LIN {X 0,Y 468.13,Z 261.484,A -85,B 0,C 180,E1 -7681.158,E2 -7681.158} C_VEL
LIN {X 0,Y 468.441,Z 256.136,A -85,B 0,C 180,E1 -7683.717,E2 -7683.717} C_VEL
LIN {X 0,Y 468.542,Z 251.799,A -85,B 0,C 180,E1 -7685.905,E2 -7685.905} C_VEL
LIN {X 0,Y 468.023,Z 247.93,A -85,B 0,C 180,E1 -7688,E2 -7688} C_VEL
LIN {X 0,Y 467.596,Z 245.244,A -85,B 0,C 180,E1 -7689.56,E2 -7689.56} C_VEL
LIN {X 0,Y 467.586,Z 245.243,A -85,B 0,C 180,E1 -7692.566,E2 -7692.566} C_VEL
LIN {X 0,Y 467.569,Z 245.245,A -85,B 0,C 180,E1 -7695.052,E2 -7695.052} C_VEL
LIN {X 0,Y 467.587,Z 245.245,A -85,B 0,C 180,E1 -7697.439,E2 -7697.439} C_VEL
LIN {X 0,Y 467.613,Z 245.241,A -85,B 0,C 180,E1 -7700.857,E2 -7700.857} C_VEL
LIN {X 0,Y 467.561,Z 245.245,A -85,B 0,C 180,E1 -7704.259,E2 -7704.259} C_VEL
LIN {X 0,Y 467.579,Z 245.243,A -85,B 0,C 180,E1 -7707.32,E2 -7707.32} C_VEL
LIN {X 0,Y 467.574,Z 245.244,A -85,B 0,C 180,E1 -7710.664,E2 -7710.664} C_VEL
LIN {X 0,Y 467.612,Z 245.239,A -85,B 0,C 180,E1 -7713.199,E2 -7713.199} C_VEL
LIN {X 0,Y 467.588,Z 245.242,A -85,B 0,C 180,E1 -7716.467,E2 -7716.467} C_VEL
LIN {X 0,Y 467.617,Z 245.239,A -85,B 0,C 180,E1 -7719.776,E2 -7719.776} C_VEL
LIN {X 0,Y 467.603,Z 245.24,A -85,B 0,C 180,E1 -7722.506,E2 -7722.506} C_VEL
LIN {X 0,Y 467.6,Z 245.242,A -85,B 0,C 180,E1 -7725.195,E2 -7725.195} C_VEL
LIN {X 0,Y 467.65,Z 245.234,A -85,B 0,C 180,E1 -7727.853,E2 -7727.853} C_VEL
LIN {X 0,Y 467.676,Z 245.232,A -85,B 0,C 180,E1 -7731.356,E2 -7731.356} C_VEL
LIN {X 0,Y 467.737,Z 245.224,A -85,B 0,C 180,E1 -7733.962,E2 -7733.962} C_VEL
LIN {X 0,Y 467.852,Z 245.21,A -85,B 0,C 180,E1 -7737.416,E2 -7737.416} C_VEL
LIN {X 0,Y 467.874,Z 245.207,A -85,B 0,C 180,E1 -7739.999,E2 -7739.999} C_VEL
LIN {X 0,Y 467.853,Z 245.211,A -85,B 0,C 180,E1 -7742.582,E2 -7742.582} C_VEL
LIN {X 0,Y 467.735,Z 245.225,A -85,B 0,C 180,E1 -7746.036,E2 -7746.036} C_VEL
LIN {X 0,Y 467.667,Z 245.234,A -85,B 0,C 180,E1 -7748.642,E2 -7748.642} C_VEL
LIN {X 0,Y 467.605,Z 245.241,A -85,B 0,C 180,E1 -7749.515,E2 -7749.515} C_VEL
LIN {X 0,Y 467.573,Z 245.747,A -85,B 0,C 180,E1 -7750.39,E2 -7750.39} C_VEL
LIN {X 0,Y 467.64,Z 248.338,A -85,B 0,C 180,E1 -7752.355,E2 -7752.355} C_VEL
LIN {X 0,Y 467.428,Z 253.066,A -85,B 0,C 180,E1 -7755.793,E2 -7755.793} C_VEL
LIN {X 0,Y 467.31,Z 257.112,A -85,B 0,C 180,E1 -7758.657,E2 -7758.657} C_VEL
LIN {X 0,Y 467.115,Z 262.092,A -85,B 0,C 180,E1 -7762.093,E2 -7762.093} C_VEL
LIN {X 0,Y 467.018,Z 267.081,A -85,B 0,C 180,E1 -7765.458,E2 -7765.458} C_VEL
LIN {X 0,Y 466.893,Z 270.645,A -85,B 0,C 180,E1 -7767.815,E2 -7767.815} C_VEL
LIN {X 0,Y 466.818,Z 275.003,A -85,B 0,C 180,E1 -7770.662,E2 -7770.662} C_VEL
LIN {X 0,Y 469.826,Z 289.237,A -85,B 0,C 180,E1 -7771.206,E2 -7771.206} C_VEL
LIN {X 0,Y 470.243,Z 292.705,A -85,B 0,C 180,E1 -7771.356,E2 -7771.356} C_VEL
LIN {X 0,Y 469.793,Z 305.072,A -85,B 0,C 180,E1 -7771.95,E2 -7771.95} C_VEL
LIN {X 0,Y 469.318,Z 316.987,A -85,B 0,C 180,E1 -7772.707,E2 -7772.707} C_VEL
LIN {X 0,Y 468.82,Z 327.819,A -85,B 0,C 180,E1 -7773.59,E2 -7773.59} C_VEL
LIN {X 0,Y 468.31,Z 338.331,A -85,B 0,C 180,E1 -7774.658,E2 -7774.658} C_VEL
LIN {X 0,Y 467.835,Z 347.892,A -85,B 0,C 180,E1 -7775.863,E2 -7775.863} C_VEL
LIN {X 0,Y 467.428,Z 356.162,A -85,B 0,C 180,E1 -7777.169,E2 -7777.169} C_VEL
LIN {X 0,Y 467.115,Z 363.055,A -85,B 0,C 180,E1 -7778.524,E2 -7778.524} C_VEL
LIN {X 0,Y 466.89,Z 368.416,A -85,B 0,C 180,E1 -7779.854,E2 -7779.854} C_VEL
LIN {X 0,Y 466.773,Z 372.503,A -85,B 0,C 180,E1 -7781.165,E2 -7781.165} C_VEL
LIN {X 0,Y 466.611,Z 375.893,A -85,B 0,C 180,E1 -7782.669,E2 -7782.669} C_VEL
LIN {X 0,Y 466.534,Z 377.66,A -85,B 0,C 180,E1 -7783.863,E2 -7783.863} C_VEL
LIN {X 0,Y 466.558,Z 378.644,A -85,B 0,C 180,E1 -7785.069,E2 -7785.069} C_VEL
LIN {X 0,Y 466.498,Z 378.866,A -85,B 0,C 180,E1 -7786.312,E2 -7786.312} C_VEL
LIN {X 0,Y 466.518,Z 378.258,A -85,B 0,C 180,E1 -7787.574,E2 -7787.574} C_VEL
LIN {X 0,Y 466.585,Z 376.759,A -85,B 0,C 180,E1 -7788.86,E2 -7788.86} C_VEL
LIN {X 0,Y 466.664,Z 374.263,A -85,B 0,C 180,E1 -7790.178,E2 -7790.178} C_VEL
LIN {X 0,Y 466.84,Z 370.669,A -85,B 0,C 180,E1 -7791.518,E2 -7791.518} C_VEL
LIN {X 0,Y 466.998,Z 365.358,A -85,B 0,C 180,E1 -7792.99,E2 -7792.99} C_VEL
LIN {X 0,Y 467.311,Z 358.15,A -85,B 0,C 180,E1 -7794.524,E2 -7794.524} C_VEL
LIN {X 0,Y 467.631,Z 350.889,A -85,B 0,C 180,E1 -7795.748,E2 -7795.748} C_VEL
LIN {X 0,Y 468.119,Z 341.5,A -85,B 0,C 180,E1 -7797.019,E2 -7797.019} C_VEL
LIN {X 0,Y 468.575,Z 331.818,A -85,B 0,C 180,E1 -7798.083,E2 -7798.083} C_VEL
LIN {X 0,Y 469.009,Z 321.069,A -85,B 0,C 180,E1 -7799.036,E2 -7799.036} C_VEL
LIN {X 0,Y 469.461,Z 309.708,A -85,B 0,C 180,E1 -7799.833,E2 -7799.833} C_VEL
LIN {X 0,Y 469.96,Z 297.671,A -85,B 0,C 180,E1 -7800.485,E2 -7800.485} C_VEL
LIN {X 0,Y 469.928,Z 290.386,A -85,B 0,C 180,E1 -7800.802,E2 -7800.802} C_VEL
LIN {X 0,Y 468.566,Z 283.472,A -85,B 0,C 180,E1 -7801.088,E2 -7801.088} C_VEL
LIN {X 0,Y 467.583,Z 280.229,A -85,B 0,C 180,E1 -7801.292,E2 -7801.292} C_VEL
LIN {X 0,Y 466.265,Z 277.641,A -85,B 0,C 180,E1 -7801.595,E2 -7801.595} C_VEL
LIN {X 0,Y 464.069,Z 274.82,A -85,B 0,C 180,E1 -7802.168,E2 -7802.168} C_VEL
LIN {X 0,Y 461.965,Z 272.984,A -85,B 0,C 180,E1 -7802.848,E2 -7802.848} C_VEL
LIN {X 0,Y 460.022,Z 271.336,A -85,B 0,C 180,E1 -7803.841,E2 -7803.841} C_VEL
LIN {X 0,Y 459.75,Z 270.573,A -85,B 0,C 180,E1 -7804.353,E2 -7804.353} C_VEL
LIN {X 0,Y 459.891,Z 265.717,A -85,B 0,C 180,E1 -7807.54,E2 -7807.54} C_VEL
LIN {X 0,Y 460.007,Z 261.493,A -85,B 0,C 180,E1 -7810.36,E2 -7810.36} C_VEL
LIN {X 0,Y 460.108,Z 257.409,A -85,B 0,C 180,E1 -7813.129,E2 -7813.129} C_VEL
LIN {X 0,Y 460.211,Z 253.466,A -85,B 0,C 180,E1 -7815.858,E2 -7815.858} C_VEL
LIN {X 0,Y 460.408,Z 249.613,A -85,B 0,C 180,E1 -7818.555,E2 -7818.555} C_VEL
LIN {X 0,Y 460.473,Z 246.127,A -85,B 0,C 180,E1 -7821.221,E2 -7821.221} C_VEL
LIN {X 0,Y 460.692,Z 246.1,A -85,B 0,C 180,E1 -7823.87,E2 -7823.87} C_VEL
LIN {X 0,Y 460.814,Z 246.084,A -85,B 0,C 180,E1 -7827.378,E2 -7827.378} C_VEL
LIN {X 0,Y 460.842,Z 246.082,A -85,B 0,C 180,E1 -7830,E2 -7830} C_VEL
LIN {X 0,Y 460.816,Z 246.086,A -85,B 0,C 180,E1 -7832.622,E2 -7832.622} C_VEL
LIN {X 0,Y 460.7,Z 246.1,A -85,B 0,C 180,E1 -7836.13,E2 -7836.13} C_VEL
LIN {X 0,Y 460.619,Z 246.11,A -85,B 0,C 180,E1 -7838.776,E2 -7838.776} C_VEL
LIN {X 0,Y 460.623,Z 246.11,A -85,B 0,C 180,E1 -7842.457,E2 -7842.457} C_VEL
LIN {X 0,Y 460.611,Z 246.111,A -85,B 0,C 180,E1 -7846.007,E2 -7846.007} C_VEL
LIN {X 0,Y 460.559,Z 246.117,A -85,B 0,C 180,E1 -7849.616,E2 -7849.616} C_VEL
LIN {X 0,Y 460.519,Z 246.122,A -85,B 0,C 180,E1 -7852.428,E2 -7852.428} C_VEL
LIN {X 0,Y 460.558,Z 246.118,A -85,B 0,C 180,E1 -7855.803,E2 -7855.803} C_VEL
LIN {X 0,Y 460.547,Z 246.12,A -85,B 0,C 180,E1 -7858.233,E2 -7858.233} C_VEL
LIN {X 0,Y 460.514,Z 246.123,A -85,B 0,C 180,E1 -7861.284,E2 -7861.284} C_VEL
LIN {X 0,Y 460.523,Z 246.121,A -85,B 0,C 180,E1 -7864.506,E2 -7864.506} C_VEL
LIN {X 0,Y 460.52,Z 246.123,A -85,B 0,C 180,E1 -7867.621,E2 -7867.621} C_VEL
LIN {X 0,Y 460.549,Z 246.118,A -85,B 0,C 180,E1 -7870.273,E2 -7870.273} C_VEL
LIN {X 0,Y 460.514,Z 246.123,A -85,B 0,C 180,E1 -7873.373,E2 -7873.373} C_VEL
LIN {X 0,Y 460.514,Z 246.123,A -85,B 0,C 180,E1 -7876.628,E2 -7876.628} C_VEL
LIN {X 0,Y 460.549,Z 246.12,A -85,B 0,C 180,E1 -7879.728,E2 -7879.728} C_VEL
LIN {X 0,Y 460.518,Z 246.122,A -85,B 0,C 180,E1 -7882.52,E2 -7882.52} C_VEL
LIN {X 0,Y 460.538,Z 246.12,A -85,B 0,C 180,E1 -7885.625,E2 -7885.625} C_VEL
LIN {X 0,Y 460.526,Z 246.122,A -85,B 0,C 180,E1 -7888.745,E2 -7888.745} C_VEL
LIN {X 0,Y 460.548,Z 246.118,A -85,B 0,C 180,E1 -7891.768,E2 -7891.768} C_VEL
LIN {X 0,Y 460.55,Z 246.12,A -85,B 0,C 180,E1 -7894.706,E2 -7894.706} C_VEL
LIN {X 0,Y 460.503,Z 246.124,A -85,B 0,C 180,E1 -7897.572,E2 -7897.572} C_VEL
LIN {X 0,Y 460.56,Z 246.117,A -85,B 0,C 180,E1 -7900.385,E2 -7900.385} C_VEL
LIN {X 0,Y 460.557,Z 246.117,A -85,B 0,C 180,E1 -7903.147,E2 -7903.147} C_VEL
LIN {X 0,Y 460.545,Z 246.117,A -85,B 0,C 180,E1 -7905.869,E2 -7905.869} C_VEL
LIN {X 0,Y 460.605,Z 246.113,A -85,B 0,C 180,E1 -7908.56,E2 -7908.56} C_VEL
LIN {X 0,Y 460.688,Z 246.101,A -85,B 0,C 180,E1 -7912.11,E2 -7912.11} C_VEL
LIN {X 0,Y 460.691,Z 246.102,A -85,B 0,C 180,E1 -7914.749,E2 -7914.749} C_VEL
LIN {X 0,Y 460.818,Z 246.084,A -85,B 0,C 180,E1 -7917.379,E2 -7917.379} C_VEL
LIN {X 0,Y 460.845,Z 246.082,A -85,B 0,C 180,E1 -7920.001,E2 -7920.001} C_VEL
LIN {X 0,Y 460.819,Z 246.085,A -85,B 0,C 180,E1 -7922.623,E2 -7922.623} C_VEL
LIN {X 0,Y 460.704,Z 246.1,A -85,B 0,C 180,E1 -7926.131,E2 -7926.131} C_VEL
LIN {X 0,Y 460.623,Z 246.109,A -85,B 0,C 180,E1 -7928.777,E2 -7928.777} C_VEL
LIN {X 0,Y 460.63,Z 246.109,A -85,B 0,C 180,E1 -7932.458,E2 -7932.458} C_VEL
LIN {X 0,Y 460.596,Z 246.113,A -85,B 0,C 180,E1 -7935.999,E2 -7935.999} C_VEL
LIN {X 0,Y 460.567,Z 246.116,A -85,B 0,C 180,E1 -7938.903,E2 -7938.903} C_VEL
LIN {X 0,Y 460.512,Z 246.124,A -85,B 0,C 180,E1 -7941.487,E2 -7941.487} C_VEL
LIN {X 0,Y 460.539,Z 246.119,A -85,B 0,C 180,E1 -7944.333,E2 -7944.333} C_VEL
LIN {X 0,Y 460.57,Z 246.117,A -85,B 0,C 180,E1 -7947.245,E2 -7947.245} C_VEL
LIN {X 0,Y 460.508,Z 246.122,A -85,B 0,C 180,E1 -7950.241,E2 -7950.241} C_VEL
LIN {X 0,Y 460.525,Z 246.123,A -85,B 0,C 180,E1 -7953.326,E2 -7953.326} C_VEL
LIN {X 0,Y 460.477,Z 246.126,A -85,B 0,C 180,E1 -7956.53,E2 -7956.53} C_VEL
LIN {X 0,Y 460.544,Z 246.119,A -85,B 0,C 180,E1 -7958.899,E2 -7958.899} C_VEL
LIN {X 0,Y 460.522,Z 246.119,A -85,B 0,C 180,E1 -7962.182,E2 -7962.182} C_VEL
LIN {X 0,Y 460.514,Z 246.123,A -85,B 0,C 180,E1 -7965.412,E2 -7965.412} C_VEL
LIN {X 0,Y 460.533,Z 246.12,A -85,B 0,C 180,E1 -7968.398,E2 -7968.398} C_VEL
LIN {X 0,Y 460.573,Z 246.124,A -85,B 0,C 180,E1 -7970.78,E2 -7970.78} C_VEL
LIN {X 0,Y 461.389,Z 251.451,A -85,B 0,C 180,E1 -7973.555,E2 -7973.555} C_VEL
LIN {X 0,Y 461.454,Z 255.827,A -85,B 0,C 180,E1 -7975.701,E2 -7975.701} C_VEL
LIN {X 0,Y 461.128,Z 262.38,A -85,B 0,C 180,E1 -7978.79,E2 -7978.79} C_VEL
LIN {X 0,Y 460.758,Z 268.954,A -85,B 0,C 180,E1 -7981.781,E2 -7981.781} C_VEL
LIN {X 0,Y 460.48,Z 276.639,A -85,B 0,C 180,E1 -7985.184,E2 -7985.184} C_VEL
LIN {X 0,Y 460.243,Z 284.73,A -85,B 0,C 180,E1 -7988.668,E2 -7988.668} C_VEL
LIN {X 0,Y 460.03,Z 292.037,A -85,B 0,C 180,E1 -7991.749,E2 -7991.749} C_VEL
LIN {X 0,Y 459.886,Z 298.398,A -85,B 0,C 180,E1 -7994.387,E2 -7994.387} C_VEL
LIN {X 0,Y 462.114,Z 312.279,A -85,B 0,C 180,E1 -7994.853,E2 -7994.853} C_VEL
LIN {X 0,Y 463.006,Z 320.585,A -85,B 0,C 180,E1 -7995.215,E2 -7995.215} C_VEL
LIN {X 0,Y 462.542,Z 332.447,A -85,B 0,C 180,E1 -7995.818,E2 -7995.818} C_VEL
LIN {X 0,Y 462.017,Z 343.944,A -85,B 0,C 180,E1 -7996.587,E2 -7996.587} C_VEL
LIN {X 0,Y 461.494,Z 355.106,A -85,B 0,C 180,E1 -7997.533,E2 -7997.533} C_VEL
LIN {X 0,Y 461.029,Z 364.99,A -85,B 0,C 180,E1 -7998.57,E2 -7998.57} C_VEL
LIN {X 0,Y 460.508,Z 373.569,A -85,B 0,C 180,E1 -7999.67,E2 -7999.67} C_VEL
LIN {X 0,Y 460.148,Z 381.911,A -85,B 0,C 180,E1 -8000.993,E2 -8000.993} C_VEL
LIN {X 0,Y 459.889,Z 388.636,A -85,B 0,C 180,E1 -8002.316,E2 -8002.316} C_VEL
LIN {X 0,Y 459.666,Z 394.798,A -85,B 0,C 180,E1 -8003.856,E2 -8003.856} C_VEL
LIN {X 0,Y 459.618,Z 398.796,A -85,B 0,C 180,E1 -8005.176,E2 -8005.176} C_VEL
LIN {X 0,Y 459.584,Z 401.745,A -85,B 0,C 180,E1 -8006.493,E2 -8006.493} C_VEL
LIN {X 0,Y 459.585,Z 403.152,A -85,B 0,C 180,E1 -8007.37,E2 -8007.37} C_VEL
LIN {X 0,Y 459.522,Z 404.758,A -85,B 0,C 180,E1 -8009.124,E2 -8009.124} C_VEL
LIN {X 0,Y 459.53,Z 404.974,A -85,B 0,C 180,E1 -8010,E2 -8010} C_VEL
LIN {X 0,Y 459.522,Z 404.753,A -85,B 0,C 180,E1 -8010.876,E2 -8010.876} C_VEL
LIN {X 0,Y 459.585,Z 403.129,A -85,B 0,C 180,E1 -8012.629,E2 -8012.629} C_VEL
LIN {X 0,Y 459.584,Z 401.718,A -85,B 0,C 180,E1 -8013.507,E2 -8013.507} C_VEL
LIN {X 0,Y 459.618,Z 398.753,A -85,B 0,C 180,E1 -8014.824,E2 -8014.824} C_VEL
LIN {X 0,Y 459.716,Z 393.705,A -85,B 0,C 180,E1 -8016.431,E2 -8016.431} C_VEL
LIN {X 0,Y 459.908,Z 387.566,A -85,B 0,C 180,E1 -8017.905,E2 -8017.905} C_VEL
LIN {X 0,Y 460.224,Z 380.617,A -85,B 0,C 180,E1 -8019.227,E2 -8019.227} C_VEL
LIN {X 0,Y 460.593,Z 371.922,A -85,B 0,C 180,E1 -8020.55,E2 -8020.55} C_VEL
LIN {X 0,Y 461.119,Z 363.024,A -85,B 0,C 180,E1 -8021.65,E2 -8021.65} C_VEL
LIN {X 0,Y 461.567,Z 352.267,A -85,B 0,C 180,E1 -8022.738,E2 -8022.738} C_VEL
LIN {X 0,Y 462.138,Z 341.06,A -85,B 0,C 180,E1 -8023.634,E2 -8023.634} C_VEL
LIN {X 0,Y 462.756,Z 328.773,A -85,B 0,C 180,E1 -8024.4,E2 -8024.4} C_VEL
LIN {X 0,Y 462.968,Z 318.49,A -85,B 0,C 180,E1 -8024.899,E2 -8024.899} C_VEL
LIN {X 0,Y 461.165,Z 305.618,A -85,B 0,C 180,E1 -8025.425,E2 -8025.425} C_VEL
LIN {X 0,Y 459.851,Z 297.977,A -85,B 0,C 180,E1 -8025.666,E2 -8025.666} C_VEL
LIN {X 0,Y 460.014,Z 290.618,A -85,B 0,C 180,E1 -8028.713,E2 -8028.713} C_VEL
LIN {X 0,Y 460.265,Z 282.926,A -85,B 0,C 180,E1 -8031.968,E2 -8031.968} C_VEL
LIN {X 0,Y 460.504,Z 275.275,A -85,B 0,C 180,E1 -8035.297,E2 -8035.297} C_VEL
LIN {X 0,Y 460.784,Z 267.719,A -85,B 0,C 180,E1 -8038.714,E2 -8038.714} C_VEL
LIN {X 0,Y 461.147,Z 262.006,A -85,B 0,C 180,E1 -8041.41,E2 -8041.41} C_VEL
LIN {X 0,Y 461.529,Z 255.372,A -85,B 0,C 180,E1 -8044.684,E2 -8044.684} C_VEL
LIN {X 0,Y 461.354,Z 251.017,A -85,B 0,C 180,E1 -8046.992,E2 -8046.992} C_VEL
LIN {X 0,Y 460.562,Z 246.12,A -85,B 0,C 180,E1 -8049.858,E2 -8049.858} C_VEL
LIN {X 0,Y 460.516,Z 246.123,A -85,B 0,C 180,E1 -8052.9,E2 -8052.9} C_VEL
LIN {X 0,Y 460.51,Z 246.125,A -85,B 0,C 180,E1 -8055.829,E2 -8055.829} C_VEL
LIN {X 0,Y 460.537,Z 246.123,A -85,B 0,C 180,E1 -8058.989,E2 -8058.989} C_VEL
LIN {X 0,Y 460.542,Z 246.121,A -85,B 0,C 180,E1 -8061.268,E2 -8061.268} C_VEL
LIN {X 0,Y 460.511,Z 246.125,A -85,B 0,C 180,E1 -8064.554,E2 -8064.554} C_VEL
LIN {X 0,Y 460.529,Z 246.122,A -85,B 0,C 180,E1 -8067.715,E2 -8067.715} C_VEL
LIN {X 0,Y 460.543,Z 246.121,A -85,B 0,C 180,E1 -8070.768,E2 -8070.768} C_VEL
LIN {X 0,Y 460.558,Z 246.118,A -85,B 0,C 180,E1 -8073.734,E2 -8073.734} C_VEL
LIN {X 0,Y 460.541,Z 246.12,A -85,B 0,C 180,E1 -8076.623,E2 -8076.623} C_VEL
LIN {X 0,Y 460.545,Z 246.12,A -85,B 0,C 180,E1 -8079.452,E2 -8079.452} C_VEL
LIN {X 0,Y 460.554,Z 246.119,A -85,B 0,C 180,E1 -8082.229,E2 -8082.229} C_VEL
LIN {X 0,Y 460.559,Z 246.118,A -85,B 0,C 180,E1 -8084.964,E2 -8084.964} C_VEL
LIN {X 0,Y 460.607,Z 246.112,A -85,B 0,C 180,E1 -8088.558,E2 -8088.558} C_VEL
LIN {X 0,Y 460.688,Z 246.102,A -85,B 0,C 180,E1 -8092.107,E2 -8092.107} C_VEL
LIN {X 0,Y 460.691,Z 246.1,A -85,B 0,C 180,E1 -8094.747,E2 -8094.747} C_VEL
LIN {X 0,Y 460.817,Z 246.086,A -85,B 0,C 180,E1 -8097.377,E2 -8097.377} C_VEL
LIN {X 0,Y 460.844,Z 246.082,A -85,B 0,C 180,E1 -8099.999,E2 -8099.999} C_VEL
LIN {X 0,Y 460.818,Z 246.088,A -85,B 0,C 180,E1 -8102.621,E2 -8102.621} C_VEL
LIN {X 0,Y 460.701,Z 246.101,A -85,B 0,C 180,E1 -8106.129,E2 -8106.129} C_VEL
LIN {X 0,Y 460.608,Z 246.114,A -85,B 0,C 180,E1 -8108.775,E2 -8108.775} C_VEL
LIN {X 0,Y 460.559,Z 246.119,A -85,B 0,C 180,E1 -8109.662,E2 -8109.662} C_VEL
LIN {X 0,Y 460.61,Z 248.118,A -85,B 0,C 180,E1 -8111.44,E2 -8111.44} C_VEL
LIN {X 0,Y 460.456,Z 251.718,A -85,B 0,C 180,E1 -8114.134,E2 -8114.134} C_VEL
LIN {X 0,Y 460.322,Z 255.431,A -85,B 0,C 180,E1 -8116.862,E2 -8116.862} C_VEL
LIN {X 0,Y 460.157,Z 259.349,A -85,B 0,C 180,E1 -8119.632,E2 -8119.632} C_VEL
LIN {X 0,Y 460.055,Z 263.387,A -85,B 0,C 180,E1 -8122.451,E2 -8122.451} C_VEL
LIN {X 0,Y 459.94,Z 268.062,A -85,B 0,C 180,E1 -8125.642,E2 -8125.642} C_VEL
LIN {X 0,Y 459.777,Z 272.019,A -85,B 0,C 180,E1 -8128.283,E2 -8128.283} C_VEL
LIN {X 0,Y 459.746,Z 275.371,A -85,B 0,C 180,E1 -8130.421,E2 -8130.421} C_VEL
LIN {X 0,Y 462.665,Z 288.74,A -85,B 0,C 180,E1 -8130.935,E2 -8130.935} C_VEL
LIN {X 0,Y 463.395,Z 293.049,A -85,B 0,C 180,E1 -8131.133,E2 -8131.133} C_VEL
LIN {X 0,Y 462.905,Z 305.934,A -85,B 0,C 180,E1 -8131.767,E2 -8131.767} C_VEL
LIN {X 0,Y 462.415,Z 317.503,A -85,B 0,C 180,E1 -8132.522,E2 -8132.522} C_VEL
LIN {X 0,Y 461.879,Z 328.845,A -85,B 0,C 180,E1 -8133.474,E2 -8133.474} C_VEL
LIN {X 0,Y 461.349,Z 338.478,A -85,B 0,C 180,E1 -8134.473,E2 -8134.473} C_VEL
LIN {X 0,Y 460.829,Z 348.261,A -85,B 0,C 180,E1 -8135.727,E2 -8135.727} C_VEL
LIN {X 0,Y 460.42,Z 356.115,A -85,B 0,C 180,E1 -8136.983,E2 -8136.983} C_VEL
LIN {X 0,Y 460.093,Z 362.404,A -85,B 0,C 180,E1 -8138.215,E2 -8138.215} C_VEL
LIN {X 0,Y 459.871,Z 368.214,A -85,B 0,C 180,E1 -8139.644,E2 -8139.644} C_VEL
LIN {X 0,Y 459.687,Z 372.748,A -85,B 0,C 180,E1 -8141.101,E2 -8141.101} C_VEL
LIN {X 0,Y 459.527,Z 376.351,A -85,B 0,C 180,E1 -8142.769,E2 -8142.769} C_VEL
LIN {X 0,Y 459.443,Z 378.086,A -85,B 0,C 180,E1 -8144.034,E2 -8144.034} C_VEL
LIN {X 0,Y 459.453,Z 378.969,A -85,B 0,C 180,E1 -8145.282,E2 -8145.282} C_VEL
LIN {X 0,Y 459.405,Z 379.03,A -85,B 0,C 180,E1 -8146.497,E2 -8146.497} C_VEL
LIN {X 0,Y 459.422,Z 378.362,A -85,B 0,C 180,E1 -8147.695,E2 -8147.695} C_VEL
LIN {X 0,Y 459.494,Z 376.99,A -85,B 0,C 180,E1 -8148.877,E2 -8148.877} C_VEL
LIN {X 0,Y 459.628,Z 373.546,A -85,B 0,C 180,E1 -8150.614,E2 -8150.614} C_VEL
LIN {X 0,Y 459.838,Z 368.499,A -85,B 0,C 180,E1 -8152.314,E2 -8152.314} C_VEL
LIN {X 0,Y 460.06,Z 362.624,A -85,B 0,C 180,E1 -8153.77,E2 -8153.77} C_VEL
LIN {X 0,Y 460.372,Z 356.11,A -85,B 0,C 180,E1 -8155.052,E2 -8155.052} C_VEL
LIN {X 0,Y 460.711,Z 349.207,A -85,B 0,C 180,E1 -8156.166,E2 -8156.166} C_VEL
LIN {X 0,Y 461.226,Z 340.032,A -85,B 0,C 180,E1 -8157.383,E2 -8157.383} C_VEL
LIN {X 0,Y 461.657,Z 329.713,A -85,B 0,C 180,E1 -8158.483,E2 -8158.483} C_VEL
LIN {X 0,Y 462.192,Z 319.286,A -85,B 0,C 180,E1 -8159.377,E2 -8159.377} C_VEL
LIN {X 0,Y 462.64,Z 307.799,A -85,B 0,C 180,E1 -8160.166,E2 -8160.166} C_VEL
LIN {X 0,Y 463.149,Z 296.398,A -85,B 0,C 180,E1 -8160.764,E2 -8160.764} C_VEL
LIN {X 0,Y 463.003,Z 291.008,A -85,B 0,C 180,E1 -8161.002,E2 -8161.002} C_VEL
LIN {X 0,Y 460.244,Z 277.687,A -85,B 0,C 180,E1 -8161.53,E2 -8161.53} C_VEL
LIN {X 0,Y 459.698,Z 274.743,A -85,B 0,C 180,E1 -8161.648,E2 -8161.648} C_VEL
LIN {X 0,Y 459.75,Z 270.573,A -85,B 0,C 180,E1 -8164.353,E2 -8164.353} C_VEL
LIN {X 0,Y 459.134,Z 269.529,A -85,B 0,C 180,E1 -8165.073,E2 -8165.073} C_VEL
LIN {X 0,Y 456.344,Z 267.993,A -85,B 0,C 180,E1 -8166.246,E2 -8166.246} C_VEL
LIN {X 0,Y 453.966,Z 266.785,A -85,B 0,C 180,E1 -8167.193,E2 -8167.193} C_VEL
LIN {X 0,Y 452.951,Z 265.789,A -85,B 0,C 180,E1 -8167.923,E2 -8167.923} C_VEL
LIN {X 0,Y 452.873,Z 265.428,A -85,B 0,C 180,E1 -8168.169,E2 -8168.169} C_VEL
LIN {X 0,Y 452.986,Z 261.029,A -85,B 0,C 180,E1 -8171.151,E2 -8171.151} C_VEL
LIN {X 0,Y 453.118,Z 256.795,A -85,B 0,C 180,E1 -8174.073,E2 -8174.073} C_VEL
LIN {X 0,Y 453.311,Z 251.774,A -85,B 0,C 180,E1 -8177.609,E2 -8177.609} C_VEL
LIN {X 0,Y 453.394,Z 247.011,A -85,B 0,C 180,E1 -8181.083,E2 -8181.083} C_VEL
LIN {X 0,Y 453.656,Z 246.976,A -85,B 0,C 180,E1 -8183.775,E2 -8183.775} C_VEL
LIN {X 0,Y 453.755,Z 246.964,A -85,B 0,C 180,E1 -8187.337,E2 -8187.337} C_VEL
LIN {X 0,Y 453.813,Z 246.958,A -85,B 0,C 180,E1 -8190,E2 -8190} C_VEL
LIN {X 0,Y 453.756,Z 246.965,A -85,B 0,C 180,E1 -8192.663,E2 -8192.663} C_VEL
LIN {X 0,Y 453.667,Z 246.976,A -85,B 0,C 180,E1 -8196.225,E2 -8196.225} C_VEL
LIN {X 0,Y 453.583,Z 246.987,A -85,B 0,C 180,E1 -8198.914,E2 -8198.914} C_VEL
LIN {X 0,Y 453.591,Z 246.987,A -85,B 0,C 180,E1 -8202.551,E2 -8202.551} C_VEL
LIN {X 0,Y 453.545,Z 246.992,A -85,B 0,C 180,E1 -8206.196,E2 -8206.196} C_VEL
LIN {X 0,Y 453.51,Z 246.994,A -85,B 0,C 180,E1 -8209.041,E2 -8209.041} C_VEL
LIN {X 0,Y 453.49,Z 246.998,A -85,B 0,C 180,E1 -8211.835,E2 -8211.835} C_VEL
LIN {X 0,Y 453.504,Z 246.995,A -85,B 0,C 180,E1 -8214.735,E2 -8214.735} C_VEL
LIN {X 0,Y 453.528,Z 246.994,A -85,B 0,C 180,E1 -8217.962,E2 -8217.962} C_VEL
LIN {X 0,Y 453.472,Z 246.999,A -85,B 0,C 180,E1 -8220.759,E2 -8220.759} C_VEL
LIN {X 0,Y 453.467,Z 247.001,A -85,B 0,C 180,E1 -8223.913,E2 -8223.913} C_VEL
LIN {X 0,Y 453.46,Z 247.002,A -85,B 0,C 180,E1 -8227.188,E2 -8227.188} C_VEL
LIN {X 0,Y 453.522,Z 246.995,A -85,B 0,C 180,E1 -8229.446,E2 -8229.446} C_VEL
LIN {X 0,Y 453.481,Z 247,A -85,B 0,C 180,E1 -8232.992,E2 -8232.992} C_VEL
LIN {X 0,Y 453.466,Z 247.001,A -85,B 0,C 180,E1 -8235.781,E2 -8235.781} C_VEL
LIN {X 0,Y 453.485,Z 246.996,A -85,B 0,C 180,E1 -8238.212,E2 -8238.212} C_VEL
LIN {X 0,Y 453.522,Z 246.993,A -85,B 0,C 180,E1 -8240.788,E2 -8240.788} C_VEL
LIN {X 0,Y 453.447,Z 247.001,A -85,B 0,C 180,E1 -8243.918,E2 -8243.918} C_VEL
LIN {X 0,Y 453.473,Z 247.002,A -85,B 0,C 180,E1 -8247.152,E2 -8247.152} C_VEL
LIN {X 0,Y 453.504,Z 246.994,A -85,B 0,C 180,E1 -8250.272,E2 -8250.272} C_VEL
LIN {X 0,Y 453.504,Z 246.996,A -85,B 0,C 180,E1 -8253.295,E2 -8253.295} C_VEL
LIN {X 0,Y 453.494,Z 246.996,A -85,B 0,C 180,E1 -8256.24,E2 -8256.24} C_VEL
LIN {X 0,Y 453.474,Z 247.001,A -85,B 0,C 180,E1 -8259.119,E2 -8259.119} C_VEL
LIN {X 0,Y 453.503,Z 246.996,A -85,B 0,C 180,E1 -8261.946,E2 -8261.946} C_VEL
LIN {X 0,Y 453.531,Z 246.993,A -85,B 0,C 180,E1 -8264.727,E2 -8264.727} C_VEL
LIN {X 0,Y 453.553,Z 246.99,A -85,B 0,C 180,E1 -8268.38,E2 -8268.38} C_VEL
LIN {X 0,Y 453.644,Z 246.978,A -85,B 0,C 180,E1 -8271.986,E2 -8271.986} C_VEL
LIN {X 0,Y 453.664,Z 246.978,A -85,B 0,C 180,E1 -8274.668,E2 -8274.668} C_VEL
LIN {X 0,Y 453.758,Z 246.963,A -85,B 0,C 180,E1 -8277.338,E2 -8277.338} C_VEL
LIN {X 0,Y 453.816,Z 246.958,A -85,B 0,C 180,E1 -8280.001,E2 -8280.001} C_VEL
LIN {X 0,Y 453.76,Z 246.964,A -85,B 0,C 180,E1 -8282.664,E2 -8282.664} C_VEL
LIN {X 0,Y 453.671,Z 246.976,A -85,B 0,C 180,E1 -8286.226,E2 -8286.226} C_VEL
LIN {X 0,Y 453.587,Z 246.985,A -85,B 0,C 180,E1 -8288.914,E2 -8288.914} C_VEL
LIN {X 0,Y 453.597,Z 246.985,A -85,B 0,C 180,E1 -8292.552,E2 -8292.552} C_VEL
LIN {X 0,Y 453.541,Z 246.993,A -85,B 0,C 180,E1 -8296.197,E2 -8296.197} C_VEL
LIN {X 0,Y 453.516,Z 246.994,A -85,B 0,C 180,E1 -8299.042,E2 -8299.042} C_VEL
LIN {X 0,Y 453.473,Z 247,A -85,B 0,C 180,E1 -8301.837,E2 -8301.837} C_VEL
LIN {X 0,Y 453.511,Z 246.994,A -85,B 0,C 180,E1 -8304.735,E2 -8304.735} C_VEL
LIN {X 0,Y 453.53,Z 246.993,A -85,B 0,C 180,E1 -8307.961,E2 -8307.961} C_VEL
LIN {X 0,Y 453.463,Z 247.002,A -85,B 0,C 180,E1 -8311.526,E2 -8311.526} C_VEL
LIN {X 0,Y 453.486,Z 246.999,A -85,B 0,C 180,E1 -8314.778,E2 -8314.778} C_VEL
LIN {X 0,Y 453.472,Z 246.999,A -85,B 0,C 180,E1 -8318.312,E2 -8318.312} C_VEL
LIN {X 0,Y 453.494,Z 246.997,A -85,B 0,C 180,E1 -8320.61,E2 -8320.61} C_VEL
LIN {X 0,Y 453.453,Z 247.003,A -85,B 0,C 180,E1 -8323.245,E2 -8323.245} C_VEL
LIN {X 0,Y 453.463,Z 247,A -85,B 0,C 180,E1 -8325.78,E2 -8325.78} C_VEL
LIN {X 0,Y 453.48,Z 246.999,A -85,B 0,C 180,E1 -8328.21,E2 -8328.21} C_VEL
LIN {X 0,Y 453.542,Z 247.089,A -85,B 0,C 180,E1 -8330.633,E2 -8330.633} C_VEL
LIN {X 0,Y 454.382,Z 252.591,A -85,B 0,C 180,E1 -8333.543,E2 -8333.543} C_VEL
LIN {X 0,Y 454.44,Z 256.79,A -85,B 0,C 180,E1 -8335.634,E2 -8335.634} C_VEL
LIN {X 0,Y 454.094,Z 263.416,A -85,B 0,C 180,E1 -8338.806,E2 -8338.806} C_VEL
LIN {X 0,Y 453.686,Z 270.341,A -85,B 0,C 180,E1 -8342.005,E2 -8342.005} C_VEL
LIN {X 0,Y 453.424,Z 277.582,A -85,B 0,C 180,E1 -8345.261,E2 -8345.261} C_VEL
LIN {X 0,Y 453.198,Z 284.982,A -85,B 0,C 180,E1 -8348.507,E2 -8348.507} C_VEL
LIN {X 0,Y 453.006,Z 291.136,A -85,B 0,C 180,E1 -8351.151,E2 -8351.151} C_VEL
LIN {X 0,Y 452.848,Z 298.23,A -85,B 0,C 180,E1 -8354.146,E2 -8354.146} C_VEL
LIN {X 0,Y 455.104,Z 312.4,A -85,B 0,C 180,E1 -8354.635,E2 -8354.635} C_VEL
LIN {X 0,Y 456.092,Z 321.46,A -85,B 0,C 180,E1 -8355.043,E2 -8355.043} C_VEL
LIN {X 0,Y 455.555,Z 333.893,A -85,B 0,C 180,E1 -8355.71,E2 -8355.71} C_VEL
LIN {X 0,Y 454.922,Z 346.469,A -85,B 0,C 180,E1 -8356.601,E2 -8356.601} C_VEL
LIN {X 0,Y 454.363,Z 357.55,A -85,B 0,C 180,E1 -8357.607,E2 -8357.607} C_VEL
LIN {X 0,Y 453.943,Z 366.544,A -85,B 0,C 180,E1 -8358.615,E2 -8358.615} C_VEL
LIN {X 0,Y 453.434,Z 374.802,A -85,B 0,C 180,E1 -8359.733,E2 -8359.733} C_VEL
LIN {X 0,Y 453.048,Z 382.901,A -85,B 0,C 180,E1 -8361.076,E2 -8361.076} C_VEL
LIN {X 0,Y 452.788,Z 389.41,A -85,B 0,C 180,E1 -8362.419,E2 -8362.419} C_VEL
LIN {X 0,Y 452.606,Z 394.575,A -85,B 0,C 180,E1 -8363.76,E2 -8363.76} C_VEL
LIN {X 0,Y 452.546,Z 398.58,A -85,B 0,C 180,E1 -8365.1,E2 -8365.1} C_VEL
LIN {X 0,Y 452.481,Z 401.534,A -85,B 0,C 180,E1 -8366.438,E2 -8366.438} C_VEL
LIN {X 0,Y 452.509,Z 402.946,A -85,B 0,C 180,E1 -8367.329,E2 -8367.329} C_VEL
LIN {X 0,Y 452.429,Z 404.555,A -85,B 0,C 180,E1 -8369.11,E2 -8369.11} C_VEL
LIN {X 0,Y 452.435,Z 404.773,A -85,B 0,C 180,E1 -8370,E2 -8370} C_VEL
LIN {X 0,Y 452.429,Z 404.555,A -85,B 0,C 180,E1 -8370.89,E2 -8370.89} C_VEL
LIN {X 0,Y 452.509,Z 402.934,A -85,B 0,C 180,E1 -8372.67,E2 -8372.67} C_VEL
LIN {X 0,Y 452.481,Z 401.523,A -85,B 0,C 180,E1 -8373.562,E2 -8373.562} C_VEL
LIN {X 0,Y 452.546,Z 398.561,A -85,B 0,C 180,E1 -8374.9,E2 -8374.9} C_VEL
LIN {X 0,Y 452.613,Z 394.012,A -85,B 0,C 180,E1 -8376.396,E2 -8376.396} C_VEL
LIN {X 0,Y 452.816,Z 388.395,A -85,B 0,C 180,E1 -8377.805,E2 -8377.805} C_VEL
LIN {X 0,Y 453.111,Z 381.672,A -85,B 0,C 180,E1 -8379.148,E2 -8379.148} C_VEL
LIN {X 0,Y 453.492,Z 373.344,A -85,B 0,C 180,E1 -8380.492,E2 -8380.492} C_VEL
LIN {X 0,Y 454.031,Z 364.814,A -85,B 0,C 180,E1 -8381.608,E2 -8381.608} C_VEL
LIN {X 0,Y 454.533,Z 355.21,A -85,B 0,C 180,E1 -8382.64,E2 -8382.64} C_VEL
LIN {X 0,Y 455.08,Z 343.915,A -85,B 0,C 180,E1 -8383.621,E2 -8383.621} C_VEL
LIN {X 0,Y 455.684,Z 332.578,A -85,B 0,C 180,E1 -8384.4,E2 -8384.4} C_VEL
LIN {X 0,Y 456.123,Z 319.728,A -85,B 0,C 180,E1 -8385.07,E2 -8385.07} C_VEL
LIN {X 0,Y 454.279,Z 306.304,A -85,B 0,C 180,E1 -8385.646,E2 -8385.646} C_VEL
LIN {X 0,Y 452.788,Z 297.751,A -85,B 0,C 180,E1 -8385.934,E2 -8385.934} C_VEL
LIN {X 0,Y 452.971,Z 290.454,A -85,B 0,C 180,E1 -8389.015,E2 -8389.015} C_VEL
LIN {X 0,Y 453.232,Z 282.787,A -85,B 0,C 180,E1 -8392.327,E2 -8392.327} C_VEL
LIN {X 0,Y 453.505,Z 275.182,A -85,B 0,C 180,E1 -8395.716,E2 -8395.716} C_VEL
LIN {X 0,Y 453.806,Z 267.668,A -85,B 0,C 180,E1 -8399.198,E2 -8399.198} C_VEL
LIN {X 0,Y 454.22,Z 261.341,A -85,B 0,C 180,E1 -8402.262,E2 -8402.262} C_VEL
LIN {X 0,Y 454.549,Z 256.001,A -85,B 0,C 180,E1 -8404.968,E2 -8404.968} C_VEL
LIN {X 0,Y 454.345,Z 252.077,A -85,B 0,C 180,E1 -8407.103,E2 -8407.103} C_VEL
LIN {X 0,Y 453.525,Z 246.996,A -85,B 0,C 180,E1 -8410.167,E2 -8410.167} C_VEL
LIN {X 0,Y 453.463,Z 247.003,A -85,B 0,C 180,E1 -8413.244,E2 -8413.244} C_VEL
LIN {X 0,Y 453.465,Z 247.003,A -85,B 0,C 180,E1 -8415.778,E2 -8415.778} C_VEL
LIN {X 0,Y 453.515,Z 246.998,A -85,B 0,C 180,E1 -8419.405,E2 -8419.405} C_VEL
LIN {X 0,Y 453.475,Z 247.001,A -85,B 0,C 180,E1 -8422.222,E2 -8422.222} C_VEL
LIN {X 0,Y 453.486,Z 246.998,A -85,B 0,C 180,E1 -8425.221,E2 -8425.221} C_VEL
LIN {X 0,Y 453.465,Z 247.002,A -85,B 0,C 180,E1 -8428.473,E2 -8428.473} C_VEL
LIN {X 0,Y 453.511,Z 246.995,A -85,B 0,C 180,E1 -8431.287,E2 -8431.287} C_VEL
LIN {X 0,Y 453.52,Z 246.994,A -85,B 0,C 180,E1 -8434.284,E2 -8434.284} C_VEL
LIN {X 0,Y 453.474,Z 247,A -85,B 0,C 180,E1 -8437.203,E2 -8437.203} C_VEL
LIN {X 0,Y 453.499,Z 246.998,A -85,B 0,C 180,E1 -8440.065,E2 -8440.065} C_VEL
LIN {X 0,Y 453.501,Z 246.997,A -85,B 0,C 180,E1 -8442.875,E2 -8442.875} C_VEL
LIN {X 0,Y 453.507,Z 246.996,A -85,B 0,C 180,E1 -8445.643,E2 -8445.643} C_VEL
LIN {X 0,Y 453.555,Z 246.991,A -85,B 0,C 180,E1 -8448.378,E2 -8448.378} C_VEL
LIN {X 0,Y 453.645,Z 246.979,A -85,B 0,C 180,E1 -8451.984,E2 -8451.984} C_VEL
LIN {X 0,Y 453.664,Z 246.976,A -85,B 0,C 180,E1 -8454.666,E2 -8454.666} C_VEL
LIN {X 0,Y 453.758,Z 246.965,A -85,B 0,C 180,E1 -8457.336,E2 -8457.336} C_VEL
LIN {X 0,Y 453.815,Z 246.958,A -85,B 0,C 180,E1 -8459.999,E2 -8459.999} C_VEL
LIN {X 0,Y 453.758,Z 246.967,A -85,B 0,C 180,E1 -8462.662,E2 -8462.662} C_VEL
LIN {X 0,Y 453.669,Z 246.977,A -85,B 0,C 180,E1 -8466.224,E2 -8466.224} C_VEL
LIN {X 0,Y 453.568,Z 246.99,A -85,B 0,C 180,E1 -8468.913,E2 -8468.913} C_VEL
LIN {X 0,Y 453.512,Z 247.065,A -85,B 0,C 180,E1 -8469.814,E2 -8469.814} C_VEL
LIN {X 0,Y 453.553,Z 250.534,A -85,B 0,C 180,E1 -8472.528,E2 -8472.528} C_VEL
LIN {X 0,Y 453.334,Z 255.196,A -85,B 0,C 180,E1 -8476.021,E2 -8476.021} C_VEL
LIN {X 0,Y 453.171,Z 259.272,A -85,B 0,C 180,E1 -8479.005,E2 -8479.005} C_VEL
LIN {X 0,Y 452.995,Z 263.325,A -85,B 0,C 180,E1 -8481.859,E2 -8481.859} C_VEL
LIN {X 0,Y 452.91,Z 267.5,A -85,B 0,C 180,E1 -8484.768,E2 -8484.768} C_VEL
LIN {X 0,Y 452.762,Z 271.92,A -85,B 0,C 180,E1 -8487.778,E2 -8487.778} C_VEL
LIN {X 0,Y 452.671,Z 275.432,A -85,B 0,C 180,E1 -8490.141,E2 -8490.141} C_VEL
LIN {X 0,Y 455.872,Z 290.094,A -85,B 0,C 180,E1 -8490.739,E2 -8490.739} C_VEL
LIN {X 0,Y 456.503,Z 293.772,A -85,B 0,C 180,E1 -8490.917,E2 -8490.917} C_VEL
LIN {X 0,Y 456.049,Z 305.997,A -85,B 0,C 180,E1 -8491.532,E2 -8491.532} C_VEL
LIN {X 0,Y 455.569,Z 317.079,A -85,B 0,C 180,E1 -8492.261,E2 -8492.261} C_VEL
LIN {X 0,Y 455.032,Z 327.176,A -85,B 0,C 180,E1 -8493.093,E2 -8493.093} C_VEL
LIN {X 0,Y 454.508,Z 336.979,A -85,B 0,C 180,E1 -8494.091,E2 -8494.091} C_VEL
LIN {X 0,Y 453.935,Z 347.009,A -85,B 0,C 180,E1 -8495.354,E2 -8495.354} C_VEL
LIN {X 0,Y 453.497,Z 354.31,A -85,B 0,C 180,E1 -8496.482,E2 -8496.482} C_VEL
LIN {X 0,Y 453.168,Z 360.948,A -85,B 0,C 180,E1 -8497.728,E2 -8497.728} C_VEL
LIN {X 0,Y 452.878,Z 366.885,A -85,B 0,C 180,E1 -8499.112,E2 -8499.112} C_VEL
LIN {X 0,Y 452.646,Z 372.069,A -85,B 0,C 180,E1 -8500.699,E2 -8500.699} C_VEL
LIN {X 0,Y 452.493,Z 375.03,A -85,B 0,C 180,E1 -8501.901,E2 -8501.901} C_VEL
LIN {X 0,Y 452.42,Z 377.206,A -85,B 0,C 180,E1 -8503.116,E2 -8503.116} C_VEL
LIN {X 0,Y 452.367,Z 378.632,A -85,B 0,C 180,E1 -8504.386,E2 -8504.386} C_VEL
LIN {X 0,Y 452.335,Z 379.253,A -85,B 0,C 180,E1 -8505.641,E2 -8505.641} C_VEL
LIN {X 0,Y 452.312,Z 379.094,A -85,B 0,C 180,E1 -8506.908,E2 -8506.908} C_VEL
LIN {X 0,Y 452.357,Z 378.082,A -85,B 0,C 180,E1 -8508.221,E2 -8508.221} C_VEL
LIN {X 0,Y 452.438,Z 376.123,A -85,B 0,C 180,E1 -8509.563,E2 -8509.563} C_VEL
LIN {X 0,Y 452.58,Z 373.126,A -85,B 0,C 180,E1 -8510.933,E2 -8510.933} C_VEL
LIN {X 0,Y 452.762,Z 368.929,A -85,B 0,C 180,E1 -8512.337,E2 -8512.337} C_VEL
LIN {X 0,Y 453.028,Z 362.828,A -85,B 0,C 180,E1 -8513.879,E2 -8513.879} C_VEL
LIN {X 0,Y 453.358,Z 355.968,A -85,B 0,C 180,E1 -8515.244,E2 -8515.244} C_VEL
LIN {X 0,Y 453.787,Z 348.46,A -85,B 0,C 180,E1 -8516.454,E2 -8516.454} C_VEL
LIN {X 0,Y 454.312,Z 338.541,A -85,B 0,C 180,E1 -8517.746,E2 -8517.746} C_VEL
LIN {X 0,Y 454.82,Z 328.215,A -85,B 0,C 180,E1 -8518.826,E2 -8518.826} C_VEL
LIN {X 0,Y 455.346,Z 317.244,A -85,B 0,C 180,E1 -8519.748,E2 -8519.748} C_VEL
LIN {X 0,Y 455.827,Z 305.813,A -85,B 0,C 180,E1 -8520.501,E2 -8520.501} C_VEL
LIN {X 0,Y 456.333,Z 293.738,A -85,B 0,C 180,E1 -8521.106,E2 -8521.106} C_VEL
LIN {X 0,Y 453.873,Z 280.922,A -85,B 0,C 180,E1 -8521.661,E2 -8521.661} C_VEL
LIN {X 0,Y 452.625,Z 274.945,A -85,B 0,C 180,E1 -8521.876,E2 -8521.876} C_VEL
LIN {X 0,Y 452.704,Z 269.862,A -85,B 0,C 180,E1 -8525.219,E2 -8525.219} C_VEL
LIN {X 0,Y 452.873,Z 265.428,A -85,B 0,C 180,E1 -8528.169,E2 -8528.169} C_VEL
LIN {X 0,Y 452.224,Z 264.405,A -85,B 0,C 180,E1 -8528.901,E2 -8528.901} C_VEL
LIN {X 0,Y 449.404,Z 262.928,A -85,B 0,C 180,E1 -8530.095,E2 -8530.095} C_VEL
LIN {X 0,Y 447.021,Z 261.772,A -85,B 0,C 180,E1 -8531.059,E2 -8531.059} C_VEL
LIN {X 0,Y 446.009,Z 260.806,A -85,B 0,C 180,E1 -8531.801,E2 -8531.801} C_VEL
LIN {X 0,Y 445.933,Z 260.453,A -85,B 0,C 180,E1 -8532.051,E2 -8532.051} C_VEL
LIN {X 0,Y 446.07,Z 257.002,A -85,B 0,C 180,E1 -8534.465,E2 -8534.465} C_VEL
LIN {X 0,Y 446.296,Z 251.797,A -85,B 0,C 180,E1 -8538.187,E2 -8538.187} C_VEL
LIN {X 0,Y 446.334,Z 248.052,A -85,B 0,C 180,E1 -8540.941,E2 -8540.941} C_VEL
LIN {X 0,Y 446.561,Z 247.862,A -85,B 0,C 180,E1 -8542.767,E2 -8542.767} C_VEL
LIN {X 0,Y 446.633,Z 247.853,A -85,B 0,C 180,E1 -8544.583,E2 -8544.583} C_VEL
LIN {X 0,Y 446.699,Z 247.843,A -85,B 0,C 180,E1 -8547.295,E2 -8547.295} C_VEL
LIN {X 0,Y 446.784,Z 247.834,A -85,B 0,C 180,E1 -8550,E2 -8550} C_VEL
LIN {X 0,Y 446.7,Z 247.844,A -85,B 0,C 180,E1 -8552.705,E2 -8552.705} C_VEL
LIN {X 0,Y 446.636,Z 247.852,A -85,B 0,C 180,E1 -8556.324,E2 -8556.324} C_VEL
LIN {X 0,Y 446.529,Z 247.864,A -85,B 0,C 180,E1 -8559.055,E2 -8559.055} C_VEL
LIN {X 0,Y 446.523,Z 247.866,A -85,B 0,C 180,E1 -8562.73,E2 -8562.73} C_VEL
LIN {X 0,Y 446.485,Z 247.871,A -85,B 0,C 180,E1 -8566.459,E2 -8566.459} C_VEL
LIN {X 0,Y 446.46,Z 247.873,A -85,B 0,C 180,E1 -8569.303,E2 -8569.303} C_VEL
LIN {X 0,Y 446.427,Z 247.879,A -85,B 0,C 180,E1 -8572.199,E2 -8572.199} C_VEL
LIN {X 0,Y 446.448,Z 247.874,A -85,B 0,C 180,E1 -8575.152,E2 -8575.152} C_VEL
LIN {X 0,Y 446.473,Z 247.873,A -85,B 0,C 180,E1 -8578.179,E2 -8578.179} C_VEL
LIN {X 0,Y 446.409,Z 247.88,A -85,B 0,C 180,E1 -8581.3,E2 -8581.3} C_VEL
LIN {X 0,Y 446.419,Z 247.877,A -85,B 0,C 180,E1 -8584.523,E2 -8584.523} C_VEL
LIN {X 0,Y 446.427,Z 247.877,A -85,B 0,C 180,E1 -8588.084,E2 -8588.084} C_VEL
LIN {X 0,Y 446.436,Z 247.876,A -85,B 0,C 180,E1 -8590.921,E2 -8590.921} C_VEL
LIN {X 0,Y 446.434,Z 247.878,A -85,B 0,C 180,E1 -8593.841,E2 -8593.841} C_VEL
LIN {X 0,Y 446.436,Z 247.875,A -85,B 0,C 180,E1 -8596.397,E2 -8596.397} C_VEL
LIN {X 0,Y 446.458,Z 247.874,A -85,B 0,C 180,E1 -8599.806,E2 -8599.806} C_VEL
LIN {X 0,Y 446.424,Z 247.877,A -85,B 0,C 180,E1 -8602.124,E2 -8602.124} C_VEL
LIN {X 0,Y 446.42,Z 247.879,A -85,B 0,C 180,E1 -8605.478,E2 -8605.478} C_VEL
LIN {X 0,Y 446.41,Z 247.881,A -85,B 0,C 180,E1 -8608.701,E2 -8608.701} C_VEL
LIN {X 0,Y 446.475,Z 247.871,A -85,B 0,C 180,E1 -8611.822,E2 -8611.822} C_VEL
LIN {X 0,Y 446.449,Z 247.876,A -85,B 0,C 180,E1 -8614.849,E2 -8614.849} C_VEL
LIN {X 0,Y 446.439,Z 247.876,A -85,B 0,C 180,E1 -8618.246,E2 -8618.246} C_VEL
LIN {X 0,Y 446.448,Z 247.874,A -85,B 0,C 180,E1 -8621.65,E2 -8621.65} C_VEL
LIN {X 0,Y 446.499,Z 247.869,A -85,B 0,C 180,E1 -8624.481,E2 -8624.481} C_VEL
LIN {X 0,Y 446.511,Z 247.867,A -85,B 0,C 180,E1 -8628.194,E2 -8628.194} C_VEL
LIN {X 0,Y 446.593,Z 247.856,A -85,B 0,C 180,E1 -8631.859,E2 -8631.859} C_VEL
LIN {X 0,Y 446.639,Z 247.853,A -85,B 0,C 180,E1 -8634.584,E2 -8634.584} C_VEL
LIN {X 0,Y 446.702,Z 247.842,A -85,B 0,C 180,E1 -8637.296,E2 -8637.296} C_VEL
LIN {X 0,Y 446.786,Z 247.834,A -85,B 0,C 180,E1 -8640.001,E2 -8640.001} C_VEL
LIN {X 0,Y 446.704,Z 247.843,A -85,B 0,C 180,E1 -8642.706,E2 -8642.706} C_VEL
LIN {X 0,Y 446.641,Z 247.851,A -85,B 0,C 180,E1 -8646.325,E2 -8646.325} C_VEL
LIN {X 0,Y 446.533,Z 247.863,A -85,B 0,C 180,E1 -8649.056,E2 -8649.056} C_VEL
LIN {X 0,Y 446.529,Z 247.864,A -85,B 0,C 180,E1 -8652.73,E2 -8652.73} C_VEL
LIN {X 0,Y 446.486,Z 247.869,A -85,B 0,C 180,E1 -8656.46,E2 -8656.46} C_VEL
LIN {X 0,Y 446.466,Z 247.873,A -85,B 0,C 180,E1 -8659.304,E2 -8659.304} C_VEL
LIN {X 0,Y 446.415,Z 247.879,A -85,B 0,C 180,E1 -8662.201,E2 -8662.201} C_VEL
LIN {X 0,Y 446.455,Z 247.875,A -85,B 0,C 180,E1 -8665.153,E2 -8665.153} C_VEL
LIN {X 0,Y 446.482,Z 247.87,A -85,B 0,C 180,E1 -8668.18,E2 -8668.18} C_VEL
LIN {X 0,Y 446.416,Z 247.88,A -85,B 0,C 180,E1 -8671.776,E2 -8671.776} C_VEL
LIN {X 0,Y 446.427,Z 247.877,A -85,B 0,C 180,E1 -8674.524,E2 -8674.524} C_VEL
LIN {X 0,Y 446.429,Z 247.876,A -85,B 0,C 180,E1 -8678.083,E2 -8678.083} C_VEL
LIN {X 0,Y 446.427,Z 247.878,A -85,B 0,C 180,E1 -8680.919,E2 -8680.919} C_VEL
LIN {X 0,Y 446.398,Z 247.881,A -85,B 0,C 180,E1 -8683.847,E2 -8683.847} C_VEL
LIN {X 0,Y 446.398,Z 247.883,A -85,B 0,C 180,E1 -8686.404,E2 -8686.404} C_VEL
LIN {X 0,Y 446.428,Z 247.877,A -85,B 0,C 180,E1 -8689.083,E2 -8689.083} C_VEL
LIN {X 0,Y 446.509,Z 248.026,A -85,B 0,C 180,E1 -8690.468,E2 -8690.468} C_VEL
LIN {X 0,Y 447.329,Z 253.363,A -85,B 0,C 180,E1 -8693.344,E2 -8693.344} C_VEL
LIN {X 0,Y 447.493,Z 256.107,A -85,B 0,C 180,E1 -8694.754,E2 -8694.754} C_VEL
LIN {X 0,Y 447.191,Z 262.094,A -85,B 0,C 180,E1 -8697.701,E2 -8697.701} C_VEL
LIN {X 0,Y 446.798,Z 268.654,A -85,B 0,C 180,E1 -8700.816,E2 -8700.816} C_VEL
LIN {X 0,Y 446.454,Z 276.314,A -85,B 0,C 180,E1 -8704.349,E2 -8704.349} C_VEL
LIN {X 0,Y 446.18,Z 283.986,A -85,B 0,C 180,E1 -8707.788,E2 -8707.788} C_VEL
LIN {X 0,Y 445.926,Z 291.364,A -85,B 0,C 180,E1 -8711.021,E2 -8711.021} C_VEL
LIN {X 0,Y 445.775,Z 298.05,A -85,B 0,C 180,E1 -8713.902,E2 -8713.902} C_VEL
LIN {X 0,Y 448.036,Z 312.053,A -85,B 0,C 180,E1 -8714.394,E2 -8714.394} C_VEL
LIN {X 0,Y 449.164,Z 322.229,A -85,B 0,C 180,E1 -8714.864,E2 -8714.864} C_VEL
LIN {X 0,Y 448.551,Z 335.269,A -85,B 0,C 180,E1 -8715.598,E2 -8715.598} C_VEL
LIN {X 0,Y 447.979,Z 346.125,A -85,B 0,C 180,E1 -8716.389,E2 -8716.389} C_VEL
LIN {X 0,Y 447.388,Z 357.245,A -85,B 0,C 180,E1 -8717.411,E2 -8717.411} C_VEL
LIN {X 0,Y 446.947,Z 366.26,A -85,B 0,C 180,E1 -8718.435,E2 -8718.435} C_VEL
LIN {X 0,Y 446.391,Z 374.534,A -85,B 0,C 180,E1 -8719.569,E2 -8719.569} C_VEL
LIN {X 0,Y 446.003,Z 382.648,A -85,B 0,C 180,E1 -8720.934,E2 -8720.934} C_VEL
LIN {X 0,Y 445.721,Z 389.171,A -85,B 0,C 180,E1 -8722.298,E2 -8722.298} C_VEL
LIN {X 0,Y 445.485,Z 395.231,A -85,B 0,C 180,E1 -8723.939,E2 -8723.939} C_VEL
LIN {X 0,Y 445.413,Z 399.436,A -85,B 0,C 180,E1 -8725.475,E2 -8725.475} C_VEL
LIN {X 0,Y 445.379,Z 401.319,A -85,B 0,C 180,E1 -8726.381,E2 -8726.381} C_VEL
LIN {X 0,Y 445.434,Z 402.738,A -85,B 0,C 180,E1 -8727.287,E2 -8727.287} C_VEL
LIN {X 0,Y 445.339,Z 404.352,A -85,B 0,C 180,E1 -8729.096,E2 -8729.096} C_VEL
LIN {X 0,Y 445.343,Z 404.573,A -85,B 0,C 180,E1 -8730,E2 -8730} C_VEL
LIN {X 0,Y 445.339,Z 404.358,A -85,B 0,C 180,E1 -8730.904,E2 -8730.904} C_VEL
LIN {X 0,Y 445.434,Z 402.739,A -85,B 0,C 180,E1 -8732.713,E2 -8732.713} C_VEL
LIN {X 0,Y 445.379,Z 401.33,A -85,B 0,C 180,E1 -8733.619,E2 -8733.619} C_VEL
LIN {X 0,Y 445.475,Z 398.371,A -85,B 0,C 180,E1 -8734.978,E2 -8734.978} C_VEL
LIN {X 0,Y 445.561,Z 392.926,A -85,B 0,C 180,E1 -8736.748,E2 -8736.748} C_VEL
LIN {X 0,Y 445.792,Z 387.198,A -85,B 0,C 180,E1 -8738.157,E2 -8738.157} C_VEL
LIN {X 0,Y 446.14,Z 380.257,A -85,B 0,C 180,E1 -8739.52,E2 -8739.52} C_VEL
LIN {X 0,Y 446.587,Z 371.581,A -85,B 0,C 180,E1 -8740.885,E2 -8740.885} C_VEL
LIN {X 0,Y 447.174,Z 362.704,A -85,B 0,C 180,E1 -8742.019,E2 -8742.019} C_VEL
LIN {X 0,Y 447.675,Z 352.398,A -85,B 0,C 180,E1 -8743.1,E2 -8743.1} C_VEL
LIN {X 0,Y 448.311,Z 340.858,A -85,B 0,C 180,E1 -8744.063,E2 -8744.063} C_VEL
LIN {X 0,Y 448.992,Z 328.658,A -85,B 0,C 180,E1 -8744.851,E2 -8744.851} C_VEL
LIN {X 0,Y 449.266,Z 321.059,A -85,B 0,C 180,E1 -8745.248,E2 -8745.248} C_VEL
LIN {X 0,Y 447.588,Z 308.259,A -85,B 0,C 180,E1 -8745.828,E2 -8745.828} C_VEL
LIN {X 0,Y 445.718,Z 297.518,A -85,B 0,C 180,E1 -8746.223,E2 -8746.223} C_VEL
LIN {X 0,Y 445.916,Z 290.301,A -85,B 0,C 180,E1 -8749.328,E2 -8749.328} C_VEL
LIN {X 0,Y 446.172,Z 282.664,A -85,B 0,C 180,E1 -8752.7,E2 -8752.7} C_VEL
LIN {X 0,Y 446.44,Z 276.166,A -85,B 0,C 180,E1 -8755.652,E2 -8755.652} C_VEL
LIN {X 0,Y 446.762,Z 268.678,A -85,B 0,C 180,E1 -8759.186,E2 -8759.186} C_VEL
LIN {X 0,Y 447.156,Z 263.099,A -85,B 0,C 180,E1 -8761.926,E2 -8761.926} C_VEL
LIN {X 0,Y 447.51,Z 258.216,A -85,B 0,C 180,E1 -8764.427,E2 -8764.427} C_VEL
LIN {X 0,Y 447.404,Z 253.949,A -85,B 0,C 180,E1 -8766.761,E2 -8766.761} C_VEL
LIN {X 0,Y 446.539,Z 248.197,A -85,B 0,C 180,E1 -8770.186,E2 -8770.186} C_VEL
LIN {X 0,Y 446.466,Z 247.876,A -85,B 0,C 180,E1 -8770.467,E2 -8770.467} C_VEL
LIN {X 0,Y 446.422,Z 247.878,A -85,B 0,C 180,E1 -8773.842,E2 -8773.842} C_VEL
LIN {X 0,Y 446.398,Z 247.883,A -85,B 0,C 180,E1 -8776.402,E2 -8776.402} C_VEL
LIN {X 0,Y 446.466,Z 247.876,A -85,B 0,C 180,E1 -8779.804,E2 -8779.804} C_VEL
LIN {X 0,Y 446.431,Z 247.878,A -85,B 0,C 180,E1 -8782.122,E2 -8782.122} C_VEL
LIN {X 0,Y 446.428,Z 247.878,A -85,B 0,C 180,E1 -8785.476,E2 -8785.476} C_VEL
LIN {X 0,Y 446.416,Z 247.88,A -85,B 0,C 180,E1 -8788.699,E2 -8788.699} C_VEL
LIN {X 0,Y 446.481,Z 247.872,A -85,B 0,C 180,E1 -8791.82,E2 -8791.82} C_VEL
LIN {X 0,Y 446.453,Z 247.875,A -85,B 0,C 180,E1 -8794.847,E2 -8794.847} C_VEL
LIN {X 0,Y 446.443,Z 247.877,A -85,B 0,C 180,E1 -8798.244,E2 -8798.244} C_VEL
LIN {X 0,Y 446.452,Z 247.875,A -85,B 0,C 180,E1 -8801.648,E2 -8801.648} C_VEL
LIN {X 0,Y 446.501,Z 247.869,A -85,B 0,C 180,E1 -8804.479,E2 -8804.479} C_VEL
LIN {X 0,Y 446.512,Z 247.868,A -85,B 0,C 180,E1 -8808.192,E2 -8808.192} C_VEL
LIN {X 0,Y 446.593,Z 247.857,A -85,B 0,C 180,E1 -8811.857,E2 -8811.857} C_VEL
LIN {X 0,Y 446.639,Z 247.851,A -85,B 0,C 180,E1 -8814.582,E2 -8814.582} C_VEL
LIN {X 0,Y 446.702,Z 247.844,A -85,B 0,C 180,E1 -8817.294,E2 -8817.294} C_VEL
LIN {X 0,Y 446.785,Z 247.833,A -85,B 0,C 180,E1 -8819.999,E2 -8819.999} C_VEL
LIN {X 0,Y 446.702,Z 247.846,A -85,B 0,C 180,E1 -8822.704,E2 -8822.704} C_VEL
LIN {X 0,Y 446.638,Z 247.852,A -85,B 0,C 180,E1 -8826.323,E2 -8826.323} C_VEL
LIN {X 0,Y 446.51,Z 247.869,A -85,B 0,C 180,E1 -8829.055,E2 -8829.055} C_VEL
LIN {X 0,Y 446.499,Z 248.318,A -85,B 0,C 180,E1 -8829.969,E2 -8829.969} C_VEL
LIN {X 0,Y 446.507,Z 251.79,A -85,B 0,C 180,E1 -8832.729,E2 -8832.729} C_VEL
LIN {X 0,Y 446.295,Z 256.259,A -85,B 0,C 180,E1 -8836.143,E2 -8836.143} C_VEL
LIN {X 0,Y 446.092,Z 260.574,A -85,B 0,C 180,E1 -8839.319,E2 -8839.319} C_VEL
LIN {X 0,Y 445.914,Z 264.629,A -85,B 0,C 180,E1 -8842.225,E2 -8842.225} C_VEL
LIN {X 0,Y 445.806,Z 268.829,A -85,B 0,C 180,E1 -8845.19,E2 -8845.19} C_VEL
LIN {X 0,Y 445.656,Z 273.256,A -85,B 0,C 180,E1 -8848.234,E2 -8848.234} C_VEL
LIN {X 0,Y 445.613,Z 275.647,A -85,B 0,C 180,E1 -8849.867,E2 -8849.867} C_VEL
LIN {X 0,Y 448.904,Z 290.56,A -85,B 0,C 180,E1 -8850.492,E2 -8850.492} C_VEL
LIN {X 0,Y 449.632,Z 296.05,A -85,B 0,C 180,E1 -8850.762,E2 -8850.762} C_VEL
LIN {X 0,Y 449.123,Z 308.286,A -85,B 0,C 180,E1 -8851.417,E2 -8851.417} C_VEL
LIN {X 0,Y 448.554,Z 319.603,A -85,B 0,C 180,E1 -8852.214,E2 -8852.214} C_VEL
LIN {X 0,Y 447.988,Z 330.343,A -85,B 0,C 180,E1 -8853.168,E2 -8853.168} C_VEL
LIN {X 0,Y 447.373,Z 340.141,A -85,B 0,C 180,E1 -8854.239,E2 -8854.239} C_VEL
LIN {X 0,Y 446.803,Z 349.984,A -85,B 0,C 180,E1 -8855.589,E2 -8855.589} C_VEL
LIN {X 0,Y 446.286,Z 358.436,A -85,B 0,C 180,E1 -8857.037,E2 -8857.037} C_VEL
LIN {X 0,Y 445.932,Z 365.196,A -85,B 0,C 180,E1 -8858.514,E2 -8858.514} C_VEL
LIN {X 0,Y 445.673,Z 369.929,A -85,B 0,C 180,E1 -8859.818,E2 -8859.818} C_VEL
LIN {X 0,Y 445.462,Z 374.513,A -85,B 0,C 180,E1 -8861.499,E2 -8861.499} C_VEL
LIN {X 0,Y 445.358,Z 376.881,A -85,B 0,C 180,E1 -8862.73,E2 -8862.73} C_VEL
LIN {X 0,Y 445.29,Z 378.512,A -85,B 0,C 180,E1 -8863.981,E2 -8863.981} C_VEL
LIN {X 0,Y 445.249,Z 379.378,A -85,B 0,C 180,E1 -8865.257,E2 -8865.257} C_VEL
LIN {X 0,Y 445.21,Z 379.418,A -85,B 0,C 180,E1 -8866.562,E2 -8866.562} C_VEL
LIN {X 0,Y 445.248,Z 378.619,A -85,B 0,C 180,E1 -8867.889,E2 -8867.889} C_VEL
LIN {X 0,Y 445.348,Z 376.185,A -85,B 0,C 180,E1 -8869.684,E2 -8869.684} C_VEL
LIN {X 0,Y 445.554,Z 372.073,A -85,B 0,C 180,E1 -8871.461,E2 -8871.461} C_VEL
LIN {X 0,Y 445.84,Z 366.304,A -85,B 0,C 180,E1 -8873.202,E2 -8873.202} C_VEL
LIN {X 0,Y 446.12,Z 359.729,A -85,B 0,C 180,E1 -8874.696,E2 -8874.696} C_VEL
LIN {X 0,Y 446.517,Z 352.463,A -85,B 0,C 180,E1 -8876.015,E2 -8876.015} C_VEL
LIN {X 0,Y 447.045,Z 343.786,A -85,B 0,C 180,E1 -8877.289,E2 -8877.289} C_VEL
LIN {X 0,Y 447.609,Z 333.144,A -85,B 0,C 180,E1 -8878.541,E2 -8878.541} C_VEL
LIN {X 0,Y 448.195,Z 321.991,A -85,B 0,C 180,E1 -8879.588,E2 -8879.588} C_VEL
LIN {X 0,Y 448.743,Z 310.413,A -85,B 0,C 180,E1 -8880.441,E2 -8880.441} C_VEL
LIN {X 0,Y 449.252,Z 299.603,A -85,B 0,C 180,E1 -8881.062,E2 -8881.062} C_VEL
LIN {X 0,Y 449.377,Z 294.049,A -85,B 0,C 180,E1 -8881.326,E2 -8881.326} C_VEL
LIN {X 0,Y 446.778,Z 280.865,A -85,B 0,C 180,E1 -8881.91,E2 -8881.91} C_VEL
LIN {X 0,Y 445.549,Z 275.123,A -85,B 0,C 180,E1 -8882.122,E2 -8882.122} C_VEL
LIN {X 0,Y 445.596,Z 271.1,A -85,B 0,C 180,E1 -8884.796,E2 -8884.796} C_VEL
LIN {X 0,Y 445.763,Z 266.685,A -85,B 0,C 180,E1 -8887.767,E2 -8887.767} C_VEL
LIN {X 0,Y 445.904,Z 261.934,A -85,B 0,C 180,E1 -8891.023,E2 -8891.023} C_VEL
LIN {X 0,Y 445.933,Z 260.453,A -85,B 0,C 180,E1 -8892.051,E2 -8892.051} C_VEL
LIN {X 0,Y 445.283,Z 259.454,A -85,B 0,C 180,E1 -8892.795,E2 -8892.795} C_VEL
LIN {X 0,Y 442.447,Z 258.039,A -85,B 0,C 180,E1 -8894.008,E2 -8894.008} C_VEL
LIN {X 0,Y 440.074,Z 256.935,A -85,B 0,C 180,E1 -8894.987,E2 -8894.987} C_VEL
LIN {X 0,Y 439.1,Z 256.001,A -85,B 0,C 180,E1 -8895.741,E2 -8895.741} C_VEL
LIN {X 0,Y 439.046,Z 255.654,A -85,B 0,C 180,E1 -8895.995,E2 -8895.995} C_VEL
LIN {X 0,Y 439.244,Z 252.9,A -85,B 0,C 180,E1 -8897.995,E2 -8897.995} C_VEL
LIN {X 0,Y 439.289,Z 249.134,A -85,B 0,C 180,E1 -8900.794,E2 -8900.794} C_VEL
LIN {X 0,Y 439.515,Z 248.739,A -85,B 0,C 180,E1 -8902.469,E2 -8902.469} C_VEL
LIN {X 0,Y 439.608,Z 248.727,A -85,B 0,C 180,E1 -8904.496,E2 -8904.496} C_VEL
LIN {X 0,Y 439.626,Z 248.724,A -85,B 0,C 180,E1 -8908.168,E2 -8908.168} C_VEL
LIN {X 0,Y 439.754,Z 248.709,A -85,B 0,C 180,E1 -8910,E2 -8910} C_VEL
LIN {X 0,Y 439.647,Z 248.723,A -85,B 0,C 180,E1 -8912.749,E2 -8912.749} C_VEL
LIN {X 0,Y 439.608,Z 248.728,A -85,B 0,C 180,E1 -8916.425,E2 -8916.425} C_VEL
LIN {X 0,Y 439.491,Z 248.74,A -85,B 0,C 180,E1 -8919.202,E2 -8919.202} C_VEL
LIN {X 0,Y 439.493,Z 248.741,A -85,B 0,C 180,E1 -8922.727,E2 -8922.727} C_VEL
LIN {X 0,Y 439.449,Z 248.748,A -85,B 0,C 180,E1 -8926.355,E2 -8926.355} C_VEL
LIN {X 0,Y 439.424,Z 248.749,A -85,B 0,C 180,E1 -8929.625,E2 -8929.625} C_VEL
LIN {X 0,Y 439.367,Z 248.756,A -85,B 0,C 180,E1 -8932.575,E2 -8932.575} C_VEL
LIN {X 0,Y 439.395,Z 248.753,A -85,B 0,C 180,E1 -8935.585,E2 -8935.585} C_VEL
LIN {X 0,Y 439.414,Z 248.749,A -85,B 0,C 180,E1 -8938.673,E2 -8938.673} C_VEL
LIN {X 0,Y 439.371,Z 248.757,A -85,B 0,C 180,E1 -8942.033,E2 -8942.033} C_VEL
LIN {X 0,Y 439.385,Z 248.755,A -85,B 0,C 180,E1 -8945.341,E2 -8945.341} C_VEL
LIN {X 0,Y 439.388,Z 248.752,A -85,B 0,C 180,E1 -8948.594,E2 -8948.594} C_VEL
LIN {X 0,Y 439.394,Z 248.754,A -85,B 0,C 180,E1 -8951.26,E2 -8951.26} C_VEL
LIN {X 0,Y 439.399,Z 248.751,A -85,B 0,C 180,E1 -8954.729,E2 -8954.729} C_VEL
LIN {X 0,Y 439.401,Z 248.752,A -85,B 0,C 180,E1 -8957.798,E2 -8957.798} C_VEL
LIN {X 0,Y 439.441,Z 248.746,A -85,B 0,C 180,E1 -8960.231,E2 -8960.231} C_VEL
LIN {X 0,Y 439.367,Z 248.756,A -85,B 0,C 180,E1 -8963.714,E2 -8963.714} C_VEL
LIN {X 0,Y 439.363,Z 248.759,A -85,B 0,C 180,E1 -8967.055,E2 -8967.055} C_VEL
LIN {X 0,Y 439.386,Z 248.753,A -85,B 0,C 180,E1 -8970.276,E2 -8970.276} C_VEL
LIN {X 0,Y 439.424,Z 248.748,A -85,B 0,C 180,E1 -8973.589,E2 -8973.589} C_VEL
LIN {X 0,Y 439.378,Z 248.755,A -85,B 0,C 180,E1 -8976.431,E2 -8976.431} C_VEL
LIN {X 0,Y 439.38,Z 248.754,A -85,B 0,C 180,E1 -8979.398,E2 -8979.398} C_VEL
LIN {X 0,Y 439.423,Z 248.75,A -85,B 0,C 180,E1 -8982.311,E2 -8982.311} C_VEL
LIN {X 0,Y 439.439,Z 248.748,A -85,B 0,C 180,E1 -8985.175,E2 -8985.175} C_VEL
LIN {X 0,Y 439.476,Z 248.744,A -85,B 0,C 180,E1 -8988.002,E2 -8988.002} C_VEL
LIN {X 0,Y 439.541,Z 248.734,A -85,B 0,C 180,E1 -8991.727,E2 -8991.727} C_VEL
LIN {X 0,Y 439.614,Z 248.727,A -85,B 0,C 180,E1 -8994.497,E2 -8994.497} C_VEL
LIN {X 0,Y 439.629,Z 248.725,A -85,B 0,C 180,E1 -8998.169,E2 -8998.169} C_VEL
LIN {X 0,Y 439.756,Z 248.709,A -85,B 0,C 180,E1 -9000.001,E2 -9000.001} C_VEL
LIN {X 0,Y 439.65,Z 248.722,A -85,B 0,C 180,E1 -9002.75,E2 -9002.75} C_VEL
LIN {X 0,Y 439.612,Z 248.727,A -85,B 0,C 180,E1 -9006.426,E2 -9006.426} C_VEL
LIN {X 0,Y 439.495,Z 248.74,A -85,B 0,C 180,E1 -9009.203,E2 -9009.203} C_VEL
LIN {X 0,Y 439.5,Z 248.739,A -85,B 0,C 180,E1 -9012.728,E2 -9012.728} C_VEL
LIN {X 0,Y 439.443,Z 248.747,A -85,B 0,C 180,E1 -9016.35,E2 -9016.35} C_VEL
LIN {X 0,Y 439.399,Z 248.754,A -85,B 0,C 180,E1 -9019.627,E2 -9019.627} C_VEL
LIN {X 0,Y 439.362,Z 248.756,A -85,B 0,C 180,E1 -9022.577,E2 -9022.577} C_VEL
LIN {X 0,Y 439.403,Z 248.753,A -85,B 0,C 180,E1 -9025.586,E2 -9025.586} C_VEL
LIN {X 0,Y 439.415,Z 248.75,A -85,B 0,C 180,E1 -9028.675,E2 -9028.675} C_VEL
LIN {X 0,Y 439.367,Z 248.756,A -85,B 0,C 180,E1 -9032.031,E2 -9032.031} C_VEL
LIN {X 0,Y 439.394,Z 248.755,A -85,B 0,C 180,E1 -9035.341,E2 -9035.341} C_VEL
LIN {X 0,Y 439.388,Z 248.754,A -85,B 0,C 180,E1 -9038.595,E2 -9038.595} C_VEL
LIN {X 0,Y 439.388,Z 248.755,A -85,B 0,C 180,E1 -9041.258,E2 -9041.258} C_VEL
LIN {X 0,Y 439.399,Z 248.753,A -85,B 0,C 180,E1 -9044.731,E2 -9044.731} C_VEL
LIN {X 0,Y 439.396,Z 248.754,A -85,B 0,C 180,E1 -9047.797,E2 -9047.797} C_VEL
LIN {X 0,Y 439.458,Z 248.83,A -85,B 0,C 180,E1 -9050.232,E2 -9050.232} C_VEL
LIN {X 0,Y 440.24,Z 253.796,A -85,B 0,C 180,E1 -9052.96,E2 -9052.96} C_VEL
LIN {X 0,Y 440.471,Z 257.588,A -85,B 0,C 180,E1 -9054.943,E2 -9054.943} C_VEL
LIN {X 0,Y 440.112,Z 264.131,A -85,B 0,C 180,E1 -9058.2,E2 -9058.2} C_VEL
LIN {X 0,Y 439.644,Z 271.106,A -85,B 0,C 180,E1 -9061.549,E2 -9061.549} C_VEL
LIN {X 0,Y 439.333,Z 278.338,A -85,B 0,C 180,E1 -9064.918,E2 -9064.918} C_VEL
LIN {X 0,Y 439.059,Z 285.99,A -85,B 0,C 180,E1 -9068.398,E2 -9068.398} C_VEL
LIN {X 0,Y 438.797,Z 293.653,A -85,B 0,C 180,E1 -9071.801,E2 -9071.801} C_VEL
LIN {X 0,Y 438.735,Z 298.078,A -85,B 0,C 180,E1 -9073.664,E2 -9073.664} C_VEL
LIN {X 0,Y 440.866,Z 311.241,A -85,B 0,C 180,E1 -9074.124,E2 -9074.124} C_VEL
LIN {X 0,Y 442.259,Z 322.906,A -85,B 0,C 180,E1 -9074.681,E2 -9074.681} C_VEL
LIN {X 0,Y 441.675,Z 334.872,A -85,B 0,C 180,E1 -9075.368,E2 -9075.368} C_VEL
LIN {X 0,Y 441.052,Z 345.762,A -85,B 0,C 180,E1 -9076.171,E2 -9076.171} C_VEL
LIN {X 0,Y 440.411,Z 356.922,A -85,B 0,C 180,E1 -9077.208,E2 -9077.208} C_VEL
LIN {X 0,Y 439.944,Z 365.957,A -85,B 0,C 180,E1 -9078.248,E2 -9078.248} C_VEL
LIN {X 0,Y 439.375,Z 374.249,A -85,B 0,C 180,E1 -9079.4,E2 -9079.4} C_VEL
LIN {X 0,Y 438.977,Z 382.38,A -85,B 0,C 180,E1 -9080.787,E2 -9080.787} C_VEL
LIN {X 0,Y 438.651,Z 388.918,A -85,B 0,C 180,E1 -9082.173,E2 -9082.173} C_VEL
LIN {X 0,Y 438.446,Z 394.345,A -85,B 0,C 180,E1 -9083.631,E2 -9083.631} C_VEL
LIN {X 0,Y 438.385,Z 398.134,A -85,B 0,C 180,E1 -9084.941,E2 -9084.941} C_VEL
LIN {X 0,Y 438.281,Z 401.1,A -85,B 0,C 180,E1 -9086.322,E2 -9086.322} C_VEL
LIN {X 0,Y 438.342,Z 402.526,A -85,B 0,C 180,E1 -9087.243,E2 -9087.243} C_VEL
LIN {X 0,Y 438.253,Z 404.147,A -85,B 0,C 180,E1 -9089.081,E2 -9089.081} C_VEL
LIN {X 0,Y 438.254,Z 404.372,A -85,B 0,C 180,E1 -9090,E2 -9090} C_VEL
LIN {X 0,Y 438.253,Z 404.162,A -85,B 0,C 180,E1 -9090.919,E2 -9090.919} C_VEL
LIN {X 0,Y 438.342,Z 402.548,A -85,B 0,C 180,E1 -9092.757,E2 -9092.757} C_VEL
LIN {X 0,Y 438.28,Z 401.141,A -85,B 0,C 180,E1 -9093.677,E2 -9093.677} C_VEL
LIN {X 0,Y 438.385,Z 398.185,A -85,B 0,C 180,E1 -9095.058,E2 -9095.058} C_VEL
LIN {X 0,Y 438.451,Z 394.184,A -85,B 0,C 180,E1 -9096.442,E2 -9096.442} C_VEL
LIN {X 0,Y 438.689,Z 388.045,A -85,B 0,C 180,E1 -9098.058,E2 -9098.058} C_VEL
LIN {X 0,Y 439.05,Z 381.341,A -85,B 0,C 180,E1 -9099.443,E2 -9099.443} C_VEL
LIN {X 0,Y 439.495,Z 373.034,A -85,B 0,C 180,E1 -9100.83,E2 -9100.83} C_VEL
LIN {X 0,Y 440.08,Z 364.54,A -85,B 0,C 180,E1 -9101.982,E2 -9101.982} C_VEL
LIN {X 0,Y 440.623,Z 354.783,A -85,B 0,C 180,E1 -9103.066,E2 -9103.066} C_VEL
LIN {X 0,Y 441.264,Z 343.748,A -85,B 0,C 180,E1 -9104.057,E2 -9104.057} C_VEL
LIN {X 0,Y 441.947,Z 332.499,A -85,B 0,C 180,E1 -9104.858,E2 -9104.858} C_VEL
LIN {X 0,Y 442.285,Z 321.119,A -85,B 0,C 180,E1 -9105.495,E2 -9105.495} C_VEL
LIN {X 0,Y 440.685,Z 308.582,A -85,B 0,C 180,E1 -9106.079,E2 -9106.079} C_VEL
LIN {X 0,Y 438.653,Z 297.294,A -85,B 0,C 180,E1 -9106.509,E2 -9106.509} C_VEL
LIN {X 0,Y 438.846,Z 290.153,A -85,B 0,C 180,E1 -9109.652,E2 -9109.652} C_VEL
LIN {X 0,Y 439.1,Z 283.625,A -85,B 0,C 180,E1 -9112.589,E2 -9112.589} C_VEL
LIN {X 0,Y 439.374,Z 277.142,A -85,B 0,C 180,E1 -9115.586,E2 -9115.586} C_VEL
LIN {X 0,Y 439.666,Z 270.732,A -85,B 0,C 180,E1 -9118.655,E2 -9118.655} C_VEL
LIN {X 0,Y 440.033,Z 265.47,A -85,B 0,C 180,E1 -9121.269,E2 -9121.269} C_VEL
LIN {X 0,Y 440.504,Z 259.255,A -85,B 0,C 180,E1 -9124.497,E2 -9124.497} C_VEL
LIN {X 0,Y 440.521,Z 256.222,A -85,B 0,C 180,E1 -9126.177,E2 -9126.177} C_VEL
LIN {X 0,Y 439.968,Z 252.208,A -85,B 0,C 180,E1 -9128.533,E2 -9128.533} C_VEL
LIN {X 0,Y 439.41,Z 248.754,A -85,B 0,C 180,E1 -9130.83,E2 -9130.83} C_VEL
LIN {X 0,Y 439.384,Z 248.755,A -85,B 0,C 180,E1 -9133.963,E2 -9133.963} C_VEL
LIN {X 0,Y 439.35,Z 248.76,A -85,B 0,C 180,E1 -9136.539,E2 -9136.539} C_VEL
LIN {X 0,Y 439.394,Z 248.756,A -85,B 0,C 180,E1 -9139.02,E2 -9139.02} C_VEL
LIN {X 0,Y 439.39,Z 248.757,A -85,B 0,C 180,E1 -9141.604,E2 -9141.604} C_VEL
LIN {X 0,Y 439.398,Z 248.754,A -85,B 0,C 180,E1 -9144.843,E2 -9144.843} C_VEL
LIN {X 0,Y 439.371,Z 248.757,A -85,B 0,C 180,E1 -9148.138,E2 -9148.138} C_VEL
LIN {X 0,Y 439.421,Z 248.75,A -85,B 0,C 180,E1 -9151.326,E2 -9151.326} C_VEL
LIN {X 0,Y 439.401,Z 248.753,A -85,B 0,C 180,E1 -9154.414,E2 -9154.414} C_VEL
LIN {X 0,Y 439.36,Z 248.758,A -85,B 0,C 180,E1 -9157.423,E2 -9157.423} C_VEL
LIN {X 0,Y 439.436,Z 248.749,A -85,B 0,C 180,E1 -9160.662,E2 -9160.662} C_VEL
LIN {X 0,Y 439.456,Z 248.747,A -85,B 0,C 180,E1 -9164.223,E2 -9164.223} C_VEL
LIN {X 0,Y 439.478,Z 248.744,A -85,B 0,C 180,E1 -9168,E2 -9168} C_VEL
LIN {X 0,Y 439.541,Z 248.736,A -85,B 0,C 180,E1 -9171.725,E2 -9171.725} C_VEL
LIN {X 0,Y 439.614,Z 248.726,A -85,B 0,C 180,E1 -9174.495,E2 -9174.495} C_VEL
LIN {X 0,Y 439.628,Z 248.725,A -85,B 0,C 180,E1 -9178.167,E2 -9178.167} C_VEL
LIN {X 0,Y 439.755,Z 248.709,A -85,B 0,C 180,E1 -9179.999,E2 -9179.999} C_VEL
LIN {X 0,Y 439.649,Z 248.725,A -85,B 0,C 180,E1 -9182.748,E2 -9182.748} C_VEL
LIN {X 0,Y 439.609,Z 248.728,A -85,B 0,C 180,E1 -9186.424,E2 -9186.424} C_VEL
LIN {X 0,Y 439.447,Z 248.749,A -85,B 0,C 180,E1 -9189.202,E2 -9189.202} C_VEL
LIN {X 0,Y 439.491,Z 250.707,A -85,B 0,C 180,E1 -9191.062,E2 -9191.062} C_VEL
LIN {X 0,Y 439.358,Z 254.256,A -85,B 0,C 180,E1 -9193.882,E2 -9193.882} C_VEL
LIN {X 0,Y 439.208,Z 257.957,A -85,B 0,C 180,E1 -9196.739,E2 -9196.739} C_VEL
LIN {X 0,Y 439.011,Z 261.879,A -85,B 0,C 180,E1 -9199.643,E2 -9199.643} C_VEL
LIN {X 0,Y 438.839,Z 265.95,A -85,B 0,C 180,E1 -9202.603,E2 -9202.603} C_VEL
LIN {X 0,Y 438.719,Z 270.188,A -85,B 0,C 180,E1 -9205.626,E2 -9205.626} C_VEL
LIN {X 0,Y 438.557,Z 274.659,A -85,B 0,C 180,E1 -9208.733,E2 -9208.733} C_VEL
LIN {X 0,Y 438.53,Z 275.892,A -85,B 0,C 180,E1 -9209.59,E2 -9209.59} C_VEL
LIN {X 0,Y 441.789,Z 290.151,A -85,B 0,C 180,E1 -9210.196,E2 -9210.196} C_VEL
LIN {X 0,Y 442.812,Z 296.547,A -85,B 0,C 180,E1 -9210.521,E2 -9210.521} C_VEL
LIN {X 0,Y 442.252,Z 309.086,A -85,B 0,C 180,E1 -9211.212,E2 -9211.212} C_VEL
LIN {X 0,Y 441.616,Z 320.783,A -85,B 0,C 180,E1 -9212.061,E2 -9212.061} C_VEL
LIN {X 0,Y 441.026,Z 331.823,A -85,B 0,C 180,E1 -9213.077,E2 -9213.077} C_VEL
LIN {X 0,Y 440.348,Z 341.872,A -85,B 0,C 180,E1 -9214.234,E2 -9214.234} C_VEL
LIN {X 0,Y 439.734,Z 351.279,A -85,B 0,C 180,E1 -9215.579,E2 -9215.579} C_VEL
LIN {X 0,Y 439.269,Z 358.617,A -85,B 0,C 180,E1 -9216.875,E2 -9216.875} C_VEL
LIN {X 0,Y 438.89,Z 365.14,A -85,B 0,C 180,E1 -9218.314,E2 -9218.314} C_VEL
LIN {X 0,Y 438.59,Z 370.608,A -85,B 0,C 180,E1 -9219.862,E2 -9219.862} C_VEL
LIN {X 0,Y 438.343,Z 375.358,A -85,B 0,C 180,E1 -9221.708,E2 -9221.708} C_VEL
LIN {X 0,Y 438.294,Z 376.783,A -85,B 0,C 180,E1 -9222.474,E2 -9222.474} C_VEL
LIN {X 0,Y 438.214,Z 378.595,A -85,B 0,C 180,E1 -9223.806,E2 -9223.806} C_VEL
LIN {X 0,Y 438.169,Z 379.518,A -85,B 0,C 180,E1 -9225.112,E2 -9225.112} C_VEL
LIN {X 0,Y 438.121,Z 379.65,A -85,B 0,C 180,E1 -9226.389,E2 -9226.389} C_VEL
LIN {X 0,Y 438.156,Z 379.046,A -85,B 0,C 180,E1 -9227.65,E2 -9227.65} C_VEL
LIN {X 0,Y 438.237,Z 377.685,A -85,B 0,C 180,E1 -9228.913,E2 -9228.913} C_VEL
LIN {X 0,Y 438.306,Z 375.232,A -85,B 0,C 180,E1 -9230.32,E2 -9230.32} C_VEL
LIN {X 0,Y 438.502,Z 371.693,A -85,B 0,C 180,E1 -9231.749,E2 -9231.749} C_VEL
LIN {X 0,Y 438.754,Z 366.855,A -85,B 0,C 180,E1 -9233.214,E2 -9233.214} C_VEL
LIN {X 0,Y 439.101,Z 359.942,A -85,B 0,C 180,E1 -9234.818,E2 -9234.818} C_VEL
LIN {X 0,Y 439.545,Z 352.166,A -85,B 0,C 180,E1 -9236.244,E2 -9236.244} C_VEL
LIN {X 0,Y 440.083,Z 343.759,A -85,B 0,C 180,E1 -9237.484,E2 -9237.484} C_VEL
LIN {X 0,Y 440.625,Z 334.103,A -85,B 0,C 180,E1 -9238.644,E2 -9238.644} C_VEL
LIN {X 0,Y 441.155,Z 324.17,A -85,B 0,C 180,E1 -9239.616,E2 -9239.616} C_VEL
LIN {X 0,Y 441.74,Z 312.656,A -85,B 0,C 180,E1 -9240.521,E2 -9240.521} C_VEL
LIN {X 0,Y 442.328,Z 300.95,A -85,B 0,C 180,E1 -9241.227,E2 -9241.227} C_VEL
LIN {X 0,Y 442.401,Z 294.667,A -85,B 0,C 180,E1 -9241.538,E2 -9241.538} C_VEL
LIN {X 0,Y 439.855,Z 281.773,A -85,B 0,C 180,E1 -9242.127,E2 -9242.127} C_VEL
LIN {X 0,Y 438.48,Z 275.312,A -85,B 0,C 180,E1 -9242.367,E2 -9242.367} C_VEL
LIN {X 0,Y 438.567,Z 270.848,A -85,B 0,C 180,E1 -9245.378,E2 -9245.378} C_VEL
LIN {X 0,Y 438.733,Z 266.449,A -85,B 0,C 180,E1 -9248.382,E2 -9248.382} C_VEL
LIN {X 0,Y 438.861,Z 262.218,A -85,B 0,C 180,E1 -9251.32,E2 -9251.32} C_VEL
LIN {X 0,Y 438.998,Z 258.133,A -85,B 0,C 180,E1 -9254.208,E2 -9254.208} C_VEL
LIN {X 0,Y 439.046,Z 255.654,A -85,B 0,C 180,E1 -9255.995,E2 -9255.995} C_VEL
LIN {X 0,Y 438.458,Z 254.684,A -85,B 0,C 180,E1 -9256.751,E2 -9256.751} C_VEL
LIN {X 0,Y 435.684,Z 253.332,A -85,B 0,C 180,E1 -9257.986,E2 -9257.986} C_VEL
LIN {X 0,Y 433.302,Z 252.277,A -85,B 0,C 180,E1 -9258.983,E2 -9258.983} C_VEL
LIN {X 0,Y 432.285,Z 251.382,A -85,B 0,C 180,E1 -9259.751,E2 -9259.751} C_VEL
LIN {X 0,Y 432.207,Z 251.05,A -85,B 0,C 180,E1 -9260.01,E2 -9260.01} C_VEL
LIN {X 0,Y 432.24,Z 250.217,A -85,B 0,C 180,E1 -9260.643,E2 -9260.643} C_VEL
LIN {X 0,Y 432.343,Z 249.629,A -85,B 0,C 180,E1 -9261.588,E2 -9261.588} C_VEL
LIN {X 0,Y 432.583,Z 249.602,A -85,B 0,C 180,E1 -9264.406,E2 -9264.406} C_VEL
LIN {X 0,Y 432.596,Z 249.6,A -85,B 0,C 180,E1 -9268.138,E2 -9268.138} C_VEL
LIN {X 0,Y 432.724,Z 249.584,A -85,B 0,C 180,E1 -9270,E2 -9270} C_VEL
LIN {X 0,Y 432.596,Z 249.601,A -85,B 0,C 180,E1 -9272.794,E2 -9272.794} C_VEL
LIN {X 0,Y 432.562,Z 249.606,A -85,B 0,C 180,E1 -9276.53,E2 -9276.53} C_VEL
LIN {X 0,Y 432.435,Z 249.619,A -85,B 0,C 180,E1 -9279.353,E2 -9279.353} C_VEL
LIN {X 0,Y 432.434,Z 249.62,A -85,B 0,C 180,E1 -9282.812,E2 -9282.812} C_VEL
LIN {X 0,Y 432.412,Z 249.623,A -85,B 0,C 180,E1 -9286.484,E2 -9286.484} C_VEL
LIN {X 0,Y 432.369,Z 249.63,A -85,B 0,C 180,E1 -9289.959,E2 -9289.959} C_VEL
LIN {X 0,Y 432.316,Z 249.632,A -85,B 0,C 180,E1 -9292.964,E2 -9292.964} C_VEL
LIN {X 0,Y 432.354,Z 249.632,A -85,B 0,C 180,E1 -9296.033,E2 -9296.033} C_VEL
LIN {X 0,Y 432.341,Z 249.631,A -85,B 0,C 180,E1 -9299.187,E2 -9299.187} C_VEL
LIN {X 0,Y 432.32,Z 249.633,A -85,B 0,C 180,E1 -9302.295,E2 -9302.295} C_VEL
LIN {X 0,Y 432.33,Z 249.632,A -85,B 0,C 180,E1 -9304.677,E2 -9304.677} C_VEL
LIN {X 0,Y 432.342,Z 249.631,A -85,B 0,C 180,E1 -9308.149,E2 -9308.149} C_VEL
LIN {X 0,Y 432.362,Z 249.631,A -85,B 0,C 180,E1 -9311.609,E2 -9311.609} C_VEL
LIN {X 0,Y 432.367,Z 249.627,A -85,B 0,C 180,E1 -9314.342,E2 -9314.342} C_VEL
LIN {X 0,Y 432.355,Z 249.631,A -85,B 0,C 180,E1 -9317.01,E2 -9317.01} C_VEL
LIN {X 0,Y 432.348,Z 249.631,A -85,B 0,C 180,E1 -9319.817,E2 -9319.817} C_VEL
LIN {X 0,Y 432.307,Z 249.637,A -85,B 0,C 180,E1 -9323.024,E2 -9323.024} C_VEL
LIN {X 0,Y 432.349,Z 249.63,A -85,B 0,C 180,E1 -9325.997,E2 -9325.997} C_VEL
LIN {X 0,Y 432.385,Z 249.625,A -85,B 0,C 180,E1 -9329.745,E2 -9329.745} C_VEL
LIN {X 0,Y 432.391,Z 249.625,A -85,B 0,C 180,E1 -9333.373,E2 -9333.373} C_VEL
LIN {X 0,Y 432.362,Z 249.628,A -85,B 0,C 180,E1 -9336.024,E2 -9336.024} C_VEL
LIN {X 0,Y 432.341,Z 249.634,A -85,B 0,C 180,E1 -9339.047,E2 -9339.047} C_VEL
LIN {X 0,Y 432.369,Z 249.628,A -85,B 0,C 180,E1 -9342.012,E2 -9342.012} C_VEL
LIN {X 0,Y 432.387,Z 249.628,A -85,B 0,C 180,E1 -9344.927,E2 -9344.927} C_VEL
LIN {X 0,Y 432.452,Z 249.617,A -85,B 0,C 180,E1 -9347.804,E2 -9347.804} C_VEL
LIN {X 0,Y 432.485,Z 249.613,A -85,B 0,C 180,E1 -9351.591,E2 -9351.591} C_VEL
LIN {X 0,Y 432.591,Z 249.602,A -85,B 0,C 180,E1 -9354.407,E2 -9354.407} C_VEL
LIN {X 0,Y 432.599,Z 249.601,A -85,B 0,C 180,E1 -9358.139,E2 -9358.139} C_VEL
LIN {X 0,Y 432.726,Z 249.585,A -85,B 0,C 180,E1 -9360.001,E2 -9360.001} C_VEL
LIN {X 0,Y 432.6,Z 249.599,A -85,B 0,C 180,E1 -9362.795,E2 -9362.795} C_VEL
LIN {X 0,Y 432.567,Z 249.605,A -85,B 0,C 180,E1 -9366.531,E2 -9366.531} C_VEL
LIN {X 0,Y 432.439,Z 249.619,A -85,B 0,C 180,E1 -9369.354,E2 -9369.354} C_VEL
LIN {X 0,Y 432.44,Z 249.618,A -85,B 0,C 180,E1 -9372.813,E2 -9372.813} C_VEL
LIN {X 0,Y 432.409,Z 249.622,A -85,B 0,C 180,E1 -9376.48,E2 -9376.48} C_VEL
LIN {X 0,Y 432.335,Z 249.634,A -85,B 0,C 180,E1 -9379.962,E2 -9379.962} C_VEL
LIN {X 0,Y 432.316,Z 249.634,A -85,B 0,C 180,E1 -9382.965,E2 -9382.965} C_VEL
LIN {X 0,Y 432.362,Z 249.629,A -85,B 0,C 180,E1 -9386.034,E2 -9386.034} C_VEL
LIN {X 0,Y 432.341,Z 249.632,A -85,B 0,C 180,E1 -9389.189,E2 -9389.189} C_VEL
LIN {X 0,Y 432.321,Z 249.633,A -85,B 0,C 180,E1 -9392.444,E2 -9392.444} C_VEL
LIN {X 0,Y 432.343,Z 249.632,A -85,B 0,C 180,E1 -9395.633,E2 -9395.633} C_VEL
LIN {X 0,Y 432.35,Z 249.63,A -85,B 0,C 180,E1 -9398.717,E2 -9398.717} C_VEL
LIN {X 0,Y 432.333,Z 249.632,A -85,B 0,C 180,E1 -9401.798,E2 -9401.798} C_VEL
LIN {X 0,Y 432.334,Z 249.632,A -85,B 0,C 180,E1 -9404.348,E2 -9404.348} C_VEL
LIN {X 0,Y 432.321,Z 249.635,A -85,B 0,C 180,E1 -9407.017,E2 -9407.017} C_VEL
LIN {X 0,Y 432.395,Z 249.718,A -85,B 0,C 180,E1 -9410.034,E2 -9410.034} C_VEL
LIN {X 0,Y 433.275,Z 255.238,A -85,B 0,C 180,E1 -9413.119,E2 -9413.119} C_VEL
LIN {X 0,Y 433.47,Z 258.517,A -85,B 0,C 180,E1 -9414.861,E2 -9414.861} C_VEL
LIN {X 0,Y 433.075,Z 265.054,A -85,B 0,C 180,E1 -9418.17,E2 -9418.17} C_VEL
LIN {X 0,Y 432.636,Z 271.476,A -85,B 0,C 180,E1 -9421.309,E2 -9421.309} C_VEL
LIN {X 0,Y 432.329,Z 278.15,A -85,B 0,C 180,E1 -9424.483,E2 -9424.483} C_VEL
LIN {X 0,Y 432.019,Z 285.805,A -85,B 0,C 180,E1 -9428.028,E2 -9428.028} C_VEL
LIN {X 0,Y 431.729,Z 293.446,A -85,B 0,C 180,E1 -9431.492,E2 -9431.492} C_VEL
LIN {X 0,Y 431.662,Z 297.825,A -85,B 0,C 180,E1 -9433.406,E2 -9433.406} C_VEL
LIN {X 0,Y 433.81,Z 311.099,A -85,B 0,C 180,E1 -9433.88,E2 -9433.88} C_VEL
LIN {X 0,Y 435.3,Z 322.365,A -85,B 0,C 180,E1 -9434.43,E2 -9434.43} C_VEL
LIN {X 0,Y 434.768,Z 334.409,A -85,B 0,C 180,E1 -9435.131,E2 -9435.131} C_VEL
LIN {X 0,Y 434.053,Z 346.554,A -85,B 0,C 180,E1 -9436.045,E2 -9436.045} C_VEL
LIN {X 0,Y 433.375,Z 357.639,A -85,B 0,C 180,E1 -9437.116,E2 -9437.116} C_VEL
LIN {X 0,Y 432.833,Z 367.422,A -85,B 0,C 180,E1 -9438.29,E2 -9438.29} C_VEL
LIN {X 0,Y 432.273,Z 375.444,A -85,B 0,C 180,E1 -9439.461,E2 -9439.461} C_VEL
LIN {X 0,Y 431.845,Z 383.313,A -85,B 0,C 180,E1 -9440.87,E2 -9440.87} C_VEL
LIN {X 0,Y 431.52,Z 390.51,A -85,B 0,C 180,E1 -9442.513,E2 -9442.513} C_VEL
LIN {X 0,Y 431.284,Z 395.627,A -85,B 0,C 180,E1 -9444.023,E2 -9444.023} C_VEL
LIN {X 0,Y 431.271,Z 398.985,A -85,B 0,C 180,E1 -9445.326,E2 -9445.326} C_VEL
LIN {X 0,Y 431.188,Z 400.878,A -85,B 0,C 180,E1 -9446.262,E2 -9446.262} C_VEL
LIN {X 0,Y 431.237,Z 402.313,A -85,B 0,C 180,E1 -9447.197,E2 -9447.197} C_VEL
LIN {X 0,Y 431.204,Z 403.323,A -85,B 0,C 180,E1 -9448.132,E2 -9448.132} C_VEL
LIN {X 0,Y 431.168,Z 404.171,A -85,B 0,C 180,E1 -9450,E2 -9450} C_VEL
LIN {X 0,Y 431.17,Z 403.967,A -85,B 0,C 180,E1 -9450.934,E2 -9450.934} C_VEL
LIN {X 0,Y 431.204,Z 403.358,A -85,B 0,C 180,E1 -9451.868,E2 -9451.868} C_VEL
LIN {X 0,Y 431.237,Z 402.358,A -85,B 0,C 180,E1 -9452.802,E2 -9452.802} C_VEL
LIN {X 0,Y 431.187,Z 400.956,A -85,B 0,C 180,E1 -9453.738,E2 -9453.738} C_VEL
LIN {X 0,Y 431.296,Z 398.007,A -85,B 0,C 180,E1 -9455.142,E2 -9455.142} C_VEL
LIN {X 0,Y 431.379,Z 394.016,A -85,B 0,C 180,E1 -9456.548,E2 -9456.548} C_VEL
LIN {X 0,Y 431.629,Z 387.891,A -85,B 0,C 180,E1 -9458.191,E2 -9458.191} C_VEL
LIN {X 0,Y 432.007,Z 381.197,A -85,B 0,C 180,E1 -9459.599,E2 -9459.599} C_VEL
LIN {X 0,Y 432.507,Z 372.9,A -85,B 0,C 180,E1 -9461.007,E2 -9461.007} C_VEL
LIN {X 0,Y 433.126,Z 364.423,A -85,B 0,C 180,E1 -9462.177,E2 -9462.177} C_VEL
LIN {X 0,Y 433.705,Z 353.888,A -85,B 0,C 180,E1 -9463.359,E2 -9463.359} C_VEL
LIN {X 0,Y 434.448,Z 342.261,A -85,B 0,C 180,E1 -9464.401,E2 -9464.401} C_VEL
LIN {X 0,Y 435.189,Z 330.616,A -85,B 0,C 180,E1 -9465.214,E2 -9465.214} C_VEL
LIN {X 0,Y 435.455,Z 322.29,A -85,B 0,C 180,E1 -9465.684,E2 -9465.684} C_VEL
LIN {X 0,Y 433.809,Z 309.324,A -85,B 0,C 180,E1 -9466.324,E2 -9466.324} C_VEL
LIN {X 0,Y 431.598,Z 297.09,A -85,B 0,C 180,E1 -9466.8,E2 -9466.8} C_VEL
LIN {X 0,Y 431.782,Z 290.005,A -85,B 0,C 180,E1 -9469.987,E2 -9469.987} C_VEL
LIN {X 0,Y 432.076,Z 283.498,A -85,B 0,C 180,E1 -9472.977,E2 -9472.977} C_VEL
LIN {X 0,Y 432.347,Z 277.051,A -85,B 0,C 180,E1 -9476.033,E2 -9476.033} C_VEL
LIN {X 0,Y 432.685,Z 270.663,A -85,B 0,C 180,E1 -9479.161,E2 -9479.161} C_VEL
LIN {X 0,Y 433.101,Z 265.426,A -85,B 0,C 180,E1 -9481.828,E2 -9481.828} C_VEL
LIN {X 0,Y 433.518,Z 260.297,A -85,B 0,C 180,E1 -9484.568,E2 -9484.568} C_VEL
LIN {X 0,Y 433.378,Z 256.256,A -85,B 0,C 180,E1 -9486.87,E2 -9486.87} C_VEL
LIN {X 0,Y 432.588,Z 250.864,A -85,B 0,C 180,E1 -9490.218,E2 -9490.218} C_VEL
LIN {X 0,Y 432.364,Z 249.632,A -85,B 0,C 180,E1 -9491.171,E2 -9491.171} C_VEL
LIN {X 0,Y 432.34,Z 249.633,A -85,B 0,C 180,E1 -9494.345,E2 -9494.345} C_VEL
LIN {X 0,Y 432.319,Z 249.637,A -85,B 0,C 180,E1 -9497.014,E2 -9497.014} C_VEL
LIN {X 0,Y 432.354,Z 249.634,A -85,B 0,C 180,E1 -9499.816,E2 -9499.816} C_VEL
LIN {X 0,Y 432.315,Z 249.636,A -85,B 0,C 180,E1 -9503.022,E2 -9503.022} C_VEL
LIN {X 0,Y 432.357,Z 249.631,A -85,B 0,C 180,E1 -9505.995,E2 -9505.995} C_VEL
LIN {X 0,Y 432.391,Z 249.627,A -85,B 0,C 180,E1 -9509.743,E2 -9509.743} C_VEL
LIN {X 0,Y 432.396,Z 249.625,A -85,B 0,C 180,E1 -9513.371,E2 -9513.371} C_VEL
LIN {X 0,Y 432.367,Z 249.63,A -85,B 0,C 180,E1 -9516.022,E2 -9516.022} C_VEL
LIN {X 0,Y 432.345,Z 249.633,A -85,B 0,C 180,E1 -9519.045,E2 -9519.045} C_VEL
LIN {X 0,Y 432.372,Z 249.63,A -85,B 0,C 180,E1 -9522.01,E2 -9522.01} C_VEL
LIN {X 0,Y 432.389,Z 249.627,A -85,B 0,C 180,E1 -9524.925,E2 -9524.925} C_VEL
LIN {X 0,Y 432.453,Z 249.618,A -85,B 0,C 180,E1 -9527.802,E2 -9527.802} C_VEL
LIN {X 0,Y 432.485,Z 249.615,A -85,B 0,C 180,E1 -9531.589,E2 -9531.589} C_VEL
LIN {X 0,Y 432.591,Z 249.602,A -85,B 0,C 180,E1 -9534.405,E2 -9534.405} C_VEL
LIN {X 0,Y 432.598,Z 249.601,A -85,B 0,C 180,E1 -9538.137,E2 -9538.137} C_VEL
LIN {X 0,Y 432.725,Z 249.585,A -85,B 0,C 180,E1 -9539.999,E2 -9539.999} C_VEL
LIN {X 0,Y 432.599,Z 249.604,A -85,B 0,C 180,E1 -9542.792,E2 -9542.792} C_VEL
LIN {X 0,Y 432.564,Z 249.606,A -85,B 0,C 180,E1 -9546.529,E2 -9546.529} C_VEL
LIN {X 0,Y 432.475,Z 249.618,A -85,B 0,C 180,E1 -9548.409,E2 -9548.409} C_VEL
LIN {X 0,Y 432.408,Z 249.713,A -85,B 0,C 180,E1 -9549.353,E2 -9549.353} C_VEL
LIN {X 0,Y 432.474,Z 253.126,A -85,B 0,C 180,E1 -9552.195,E2 -9552.195} C_VEL
LIN {X 0,Y 432.248,Z 257.994,A -85,B 0,C 180,E1 -9556.045,E2 -9556.045} C_VEL
LIN {X 0,Y 431.995,Z 262.311,A -85,B 0,C 180,E1 -9559.341,E2 -9559.341} C_VEL
LIN {X 0,Y 431.773,Z 267.27,A -85,B 0,C 180,E1 -9562.993,E2 -9562.993} C_VEL
LIN {X 0,Y 431.645,Z 271.55,A -85,B 0,C 180,E1 -9566.078,E2 -9566.078} C_VEL
LIN {X 0,Y 431.501,Z 276.1,A -85,B 0,C 180,E1 -9569.282,E2 -9569.282} C_VEL
LIN {X 0,Y 434.832,Z 290.726,A -85,B 0,C 180,E1 -9569.934,E2 -9569.934} C_VEL
LIN {X 0,Y 435.973,Z 297.85,A -85,B 0,C 180,E1 -9570.31,E2 -9570.31} C_VEL
LIN {X 0,Y 435.39,Z 310.024,A -85,B 0,C 180,E1 -9571.01,E2 -9571.01} C_VEL
LIN {X 0,Y 434.702,Z 322.397,A -85,B 0,C 180,E1 -9571.942,E2 -9571.942} C_VEL
LIN {X 0,Y 434.037,Z 333.435,A -85,B 0,C 180,E1 -9573.007,E2 -9573.007} C_VEL
LIN {X 0,Y 433.323,Z 343.32,A -85,B 0,C 180,E1 -9574.194,E2 -9574.194} C_VEL
LIN {X 0,Y 432.776,Z 351.538,A -85,B 0,C 180,E1 -9575.404,E2 -9575.404} C_VEL
LIN {X 0,Y 432.273,Z 358.7,A -85,B 0,C 180,E1 -9576.689,E2 -9576.689} C_VEL
LIN {X 0,Y 431.833,Z 365.449,A -85,B 0,C 180,E1 -9578.201,E2 -9578.201} C_VEL
LIN {X 0,Y 431.603,Z 369.828,A -85,B 0,C 180,E1 -9579.422,E2 -9579.422} C_VEL
LIN {X 0,Y 431.392,Z 373.371,A -85,B 0,C 180,E1 -9580.665,E2 -9580.665} C_VEL
LIN {X 0,Y 431.228,Z 376.137,A -85,B 0,C 180,E1 -9581.927,E2 -9581.927} C_VEL
LIN {X 0,Y 431.162,Z 378.149,A -85,B 0,C 180,E1 -9583.203,E2 -9583.203} C_VEL
LIN {X 0,Y 431.091,Z 379.428,A -85,B 0,C 180,E1 -9584.507,E2 -9584.507} C_VEL
LIN {X 0,Y 431.062,Z 379.894,A -85,B 0,C 180,E1 -9585.836,E2 -9585.836} C_VEL
LIN {X 0,Y 431.015,Z 379.545,A -85,B 0,C 180,E1 -9587.2,E2 -9587.2} C_VEL
LIN {X 0,Y 431.118,Z 378.332,A -85,B 0,C 180,E1 -9588.578,E2 -9588.578} C_VEL
LIN {X 0,Y 431.182,Z 376.152,A -85,B 0,C 180,E1 -9590,E2 -9590} C_VEL
LIN {X 0,Y 431.429,Z 372.078,A -85,B 0,C 180,E1 -9591.756,E2 -9591.756} C_VEL
LIN {X 0,Y 431.753,Z 366.141,A -85,B 0,C 180,E1 -9593.55,E2 -9593.55} C_VEL
LIN {X 0,Y 432.128,Z 359.417,A -85,B 0,C 180,E1 -9595.094,E2 -9595.094} C_VEL
LIN {X 0,Y 432.558,Z 351.909,A -85,B 0,C 180,E1 -9596.468,E2 -9596.468} C_VEL
LIN {X 0,Y 433.193,Z 343.057,A -85,B 0,C 180,E1 -9597.768,E2 -9597.768} C_VEL
LIN {X 0,Y 433.757,Z 332.771,A -85,B 0,C 180,E1 -9598.997,E2 -9598.997} C_VEL
LIN {X 0,Y 434.366,Z 322.158,A -85,B 0,C 180,E1 -9600.011,E2 -9600.011} C_VEL
LIN {X 0,Y 435.02,Z 309.85,A -85,B 0,C 180,E1 -9600.935,E2 -9600.935} C_VEL
LIN {X 0,Y 435.658,Z 297.714,A -85,B 0,C 180,E1 -9601.63,E2 -9601.63} C_VEL
LIN {X 0,Y 433.565,Z 285.66,A -85,B 0,C 180,E1 -9602.224,E2 -9602.224} C_VEL
LIN {X 0,Y 431.406,Z 275.486,A -85,B 0,C 180,E1 -9602.632,E2 -9602.632} C_VEL
LIN {X 0,Y 431.527,Z 270.594,A -85,B 0,C 180,E1 -9605.974,E2 -9605.974} C_VEL
LIN {X 0,Y 431.668,Z 266.212,A -85,B 0,C 180,E1 -9609.012,E2 -9609.012} C_VEL
LIN {X 0,Y 431.806,Z 262.011,A -85,B 0,C 180,E1 -9611.987,E2 -9611.987} C_VEL
LIN {X 0,Y 431.928,Z 257.941,A -85,B 0,C 180,E1 -9614.91,E2 -9614.91} C_VEL
LIN {X 0,Y 432.172,Z 254.002,A -85,B 0,C 180,E1 -9617.796,E2 -9617.796} C_VEL
LIN {X 0,Y 432.207,Z 251.05,A -85,B 0,C 180,E1 -9620.01,E2 -9620.01} C_VEL
LIN {X 0,Y 431.572,Z 250.327,A -85,B 0,C 180,E1 -9620.782,E2 -9620.782} C_VEL
LIN {X 0,Y 428.829,Z 250.089,A -85,B 0,C 180,E1 -9622.05,E2 -9622.05} C_VEL
LIN {X 0,Y 426.527,Z 250.357,A -85,B 0,C 180,E1 -9623.078,E2 -9623.078} C_VEL
LIN {X 0,Y 425.578,Z 250.474,A -85,B 0,C 180,E1 -9623.871,E2 -9623.871} C_VEL
LIN {X 0,Y 425.521,Z 250.48,A -85,B 0,C 180,E1 -9624.139,E2 -9624.139} C_VEL
LIN {X 0,Y 425.565,Z 250.475,A -85,B 0,C 180,E1 -9628.107,E2 -9628.107} C_VEL
LIN {X 0,Y 425.694,Z 250.46,A -85,B 0,C 180,E1 -9630,E2 -9630} C_VEL
LIN {X 0,Y 425.548,Z 250.479,A -85,B 0,C 180,E1 -9632.84,E2 -9632.84} C_VEL
LIN {X 0,Y 425.52,Z 250.483,A -85,B 0,C 180,E1 -9636.639,E2 -9636.639} C_VEL
LIN {X 0,Y 425.394,Z 250.496,A -85,B 0,C 180,E1 -9639.509,E2 -9639.509} C_VEL
LIN {X 0,Y 425.393,Z 250.496,A -85,B 0,C 180,E1 -9642.91,E2 -9642.91} C_VEL
LIN {X 0,Y 425.359,Z 250.501,A -85,B 0,C 180,E1 -9646.609,E2 -9646.609} C_VEL
LIN {X 0,Y 425.351,Z 250.502,A -85,B 0,C 180,E1 -9649.649,E2 -9649.649} C_VEL
LIN {X 0,Y 425.301,Z 250.507,A -85,B 0,C 180,E1 -9653.365,E2 -9653.365} C_VEL
LIN {X 0,Y 425.338,Z 250.502,A -85,B 0,C 180,E1 -9656.845,E2 -9656.845} C_VEL
LIN {X 0,Y 425.307,Z 250.51,A -85,B 0,C 180,E1 -9659.718,E2 -9659.718} C_VEL
LIN {X 0,Y 425.273,Z 250.511,A -85,B 0,C 180,E1 -9663.048,E2 -9663.048} C_VEL
LIN {X 0,Y 425.274,Z 250.512,A -85,B 0,C 180,E1 -9665.93,E2 -9665.93} C_VEL
LIN {X 0,Y 425.302,Z 250.508,A -85,B 0,C 180,E1 -9669.047,E2 -9669.047} C_VEL
LIN {X 0,Y 425.321,Z 250.505,A -85,B 0,C 180,E1 -9672.646,E2 -9672.646} C_VEL
LIN {X 0,Y 425.308,Z 250.507,A -85,B 0,C 180,E1 -9676.052,E2 -9676.052} C_VEL
LIN {X 0,Y 425.299,Z 250.507,A -85,B 0,C 180,E1 -9678.626,E2 -9678.626} C_VEL
LIN {X 0,Y 425.314,Z 250.509,A -85,B 0,C 180,E1 -9681.105,E2 -9681.105} C_VEL
LIN {X 0,Y 425.29,Z 250.509,A -85,B 0,C 180,E1 -9684.665,E2 -9684.665} C_VEL
LIN {X 0,Y 425.256,Z 250.512,A -85,B 0,C 180,E1 -9688.074,E2 -9688.074} C_VEL
LIN {X 0,Y 425.328,Z 250.506,A -85,B 0,C 180,E1 -9691.369,E2 -9691.369} C_VEL
LIN {X 0,Y 425.286,Z 250.511,A -85,B 0,C 180,E1 -9694.556,E2 -9694.556} C_VEL
LIN {X 0,Y 425.279,Z 250.51,A -85,B 0,C 180,E1 -9697.662,E2 -9697.662} C_VEL
LIN {X 0,Y 425.353,Z 250.504,A -85,B 0,C 180,E1 -9700.705,E2 -9700.705} C_VEL
LIN {X 0,Y 425.38,Z 250.497,A -85,B 0,C 180,E1 -9703.689,E2 -9703.689} C_VEL
LIN {X 0,Y 425.404,Z 250.495,A -85,B 0,C 180,E1 -9707.599,E2 -9707.599} C_VEL
LIN {X 0,Y 425.435,Z 250.49,A -85,B 0,C 180,E1 -9711.451,E2 -9711.451} C_VEL
LIN {X 0,Y 425.547,Z 250.479,A -85,B 0,C 180,E1 -9714.314,E2 -9714.314} C_VEL
LIN {X 0,Y 425.569,Z 250.476,A -85,B 0,C 180,E1 -9718.108,E2 -9718.108} C_VEL
LIN {X 0,Y 425.696,Z 250.461,A -85,B 0,C 180,E1 -9720.001,E2 -9720.001} C_VEL
LIN {X 0,Y 425.552,Z 250.477,A -85,B 0,C 180,E1 -9722.841,E2 -9722.841} C_VEL
LIN {X 0,Y 425.525,Z 250.481,A -85,B 0,C 180,E1 -9726.64,E2 -9726.64} C_VEL
LIN {X 0,Y 425.398,Z 250.497,A -85,B 0,C 180,E1 -9729.51,E2 -9729.51} C_VEL
LIN {X 0,Y 425.4,Z 250.495,A -85,B 0,C 180,E1 -9732.911,E2 -9732.911} C_VEL
LIN {X 0,Y 425.358,Z 250.5,A -85,B 0,C 180,E1 -9736.606,E2 -9736.606} C_VEL
LIN {X 0,Y 425.325,Z 250.507,A -85,B 0,C 180,E1 -9739.637,E2 -9739.637} C_VEL
LIN {X 0,Y 425.304,Z 250.509,A -85,B 0,C 180,E1 -9743.366,E2 -9743.366} C_VEL
LIN {X 0,Y 425.345,Z 250.501,A -85,B 0,C 180,E1 -9746.845,E2 -9746.845} C_VEL
LIN {X 0,Y 425.289,Z 250.511,A -85,B 0,C 180,E1 -9749.721,E2 -9749.721} C_VEL
LIN {X 0,Y 425.28,Z 250.511,A -85,B 0,C 180,E1 -9753.049,E2 -9753.049} C_VEL
LIN {X 0,Y 425.282,Z 250.51,A -85,B 0,C 180,E1 -9755.93,E2 -9755.93} C_VEL
LIN {X 0,Y 425.3,Z 250.51,A -85,B 0,C 180,E1 -9759.045,E2 -9759.045} C_VEL
LIN {X 0,Y 425.274,Z 250.511,A -85,B 0,C 180,E1 -9762.654,E2 -9762.654} C_VEL
LIN {X 0,Y 425.262,Z 250.513,A -85,B 0,C 180,E1 -9766.045,E2 -9766.045} C_VEL
LIN {X 0,Y 425.294,Z 250.509,A -85,B 0,C 180,E1 -9769.479,E2 -9769.479} C_VEL
LIN {X 0,Y 425.374,Z 250.679,A -85,B 0,C 180,E1 -9769.883,E2 -9769.883} C_VEL
LIN {X 0,Y 426.24,Z 256.166,A -85,B 0,C 180,E1 -9773,E2 -9773} C_VEL
LIN {X 0,Y 426.378,Z 260.83,A -85,B 0,C 180,E1 -9775.504,E2 -9775.504} C_VEL
LIN {X 0,Y 426.058,Z 265.98,A -85,B 0,C 180,E1 -9778.14,E2 -9778.14} C_VEL
LIN {X 0,Y 425.569,Z 272.511,A -85,B 0,C 180,E1 -9781.386,E2 -9781.386} C_VEL
LIN {X 0,Y 425.274,Z 279.064,A -85,B 0,C 180,E1 -9784.554,E2 -9784.554} C_VEL
LIN {X 0,Y 424.945,Z 286.037,A -85,B 0,C 180,E1 -9787.846,E2 -9787.846} C_VEL
LIN {X 0,Y 424.683,Z 293.236,A -85,B 0,C 180,E1 -9791.174,E2 -9791.174} C_VEL
LIN {X 0,Y 424.584,Z 297.551,A -85,B 0,C 180,E1 -9793.137,E2 -9793.137} C_VEL
LIN {X 0,Y 426.875,Z 311.292,A -85,B 0,C 180,E1 -9793.645,E2 -9793.645} C_VEL
LIN {X 0,Y 428.415,Z 324.057,A -85,B 0,C 180,E1 -9794.296,E2 -9794.296} C_VEL
LIN {X 0,Y 427.776,Z 335.684,A -85,B 0,C 180,E1 -9795.004,E2 -9795.004} C_VEL
LIN {X 0,Y 427.127,Z 346.298,A -85,B 0,C 180,E1 -9795.829,E2 -9795.829} C_VEL
LIN {X 0,Y 426.418,Z 357.267,A -85,B 0,C 180,E1 -9796.902,E2 -9796.902} C_VEL
LIN {X 0,Y 425.847,Z 367.079,A -85,B 0,C 180,E1 -9798.095,E2 -9798.095} C_VEL
LIN {X 0,Y 425.256,Z 375.125,A -85,B 0,C 180,E1 -9799.285,E2 -9799.285} C_VEL
LIN {X 0,Y 424.803,Z 383.024,A -85,B 0,C 180,E1 -9800.717,E2 -9800.717} C_VEL
LIN {X 0,Y 424.526,Z 388.38,A -85,B 0,C 180,E1 -9801.911,E2 -9801.911} C_VEL
LIN {X 0,Y 424.303,Z 393.608,A -85,B 0,C 180,E1 -9803.342,E2 -9803.342} C_VEL
LIN {X 0,Y 424.209,Z 397.66,A -85,B 0,C 180,E1 -9804.772,E2 -9804.772} C_VEL
LIN {X 0,Y 424.099,Z 400.647,A -85,B 0,C 180,E1 -9806.199,E2 -9806.199} C_VEL
LIN {X 0,Y 424.133,Z 402.093,A -85,B 0,C 180,E1 -9807.151,E2 -9807.151} C_VEL
LIN {X 0,Y 424.13,Z 403.11,A -85,B 0,C 180,E1 -9808.101,E2 -9808.101} C_VEL
LIN {X 0,Y 424.085,Z 403.968,A -85,B 0,C 180,E1 -9810,E2 -9810} C_VEL
LIN {X 0,Y 424.089,Z 403.774,A -85,B 0,C 180,E1 -9810.949,E2 -9810.949} C_VEL
LIN {X 0,Y 424.13,Z 403.17,A -85,B 0,C 180,E1 -9811.899,E2 -9811.899} C_VEL
LIN {X 0,Y 424.132,Z 402.173,A -85,B 0,C 180,E1 -9812.849,E2 -9812.849} C_VEL
LIN {X 0,Y 424.099,Z 400.775,A -85,B 0,C 180,E1 -9813.801,E2 -9813.801} C_VEL
LIN {X 0,Y 424.208,Z 397.833,A -85,B 0,C 180,E1 -9815.228,E2 -9815.228} C_VEL
LIN {X 0,Y 424.303,Z 393.85,A -85,B 0,C 180,E1 -9816.658,E2 -9816.658} C_VEL
LIN {X 0,Y 424.585,Z 387.738,A -85,B 0,C 180,E1 -9818.327,E2 -9818.327} C_VEL
LIN {X 0,Y 424.979,Z 381.052,A -85,B 0,C 180,E1 -9819.759,E2 -9819.759} C_VEL
LIN {X 0,Y 425.497,Z 372.765,A -85,B 0,C 180,E1 -9821.19,E2 -9821.19} C_VEL
LIN {X 0,Y 426.18,Z 364.305,A -85,B 0,C 180,E1 -9822.379,E2 -9822.379} C_VEL
LIN {X 0,Y 426.729,Z 354.61,A -85,B 0,C 180,E1 -9823.499,E2 -9823.499} C_VEL
LIN {X 0,Y 427.457,Z 343.651,A -85,B 0,C 180,E1 -9824.52,E2 -9824.52} C_VEL
LIN {X 0,Y 428.234,Z 332.51,A -85,B 0,C 180,E1 -9825.345,E2 -9825.345} C_VEL
LIN {X 0,Y 428.535,Z 322.433,A -85,B 0,C 180,E1 -9825.944,E2 -9825.944} C_VEL
LIN {X 0,Y 426.935,Z 309.751,A -85,B 0,C 180,E1 -9826.594,E2 -9826.594} C_VEL
LIN {X 0,Y 424.534,Z 296.907,A -85,B 0,C 180,E1 -9827.101,E2 -9827.101} C_VEL
LIN {X 0,Y 424.756,Z 289.873,A -85,B 0,C 180,E1 -9830.332,E2 -9830.332} C_VEL
LIN {X 0,Y 425.04,Z 283.394,A -85,B 0,C 180,E1 -9833.38,E2 -9833.38} C_VEL
LIN {X 0,Y 425.365,Z 276.974,A -85,B 0,C 180,E1 -9836.493,E2 -9836.493} C_VEL
LIN {X 0,Y 425.846,Z 269.579,A -85,B 0,C 180,E1 -9840.222,E2 -9840.222} C_VEL
LIN {X 0,Y 426.219,Z 264.401,A -85,B 0,C 180,E1 -9842.965,E2 -9842.965} C_VEL
LIN {X 0,Y 426.526,Z 260.327,A -85,B 0,C 180,E1 -9845.218,E2 -9845.218} C_VEL
LIN {X 0,Y 426.229,Z 256.174,A -85,B 0,C 180,E1 -9847.677,E2 -9847.677} C_VEL
LIN {X 0,Y 425.536,Z 251.706,A -85,B 0,C 180,E1 -9850.559,E2 -9850.559} C_VEL
LIN {X 0,Y 425.31,Z 250.51,A -85,B 0,C 180,E1 -9851.518,E2 -9851.518} C_VEL
LIN {X 0,Y 425.285,Z 250.511,A -85,B 0,C 180,E1 -9855.282,E2 -9855.282} C_VEL
LIN {X 0,Y 425.303,Z 250.512,A -85,B 0,C 180,E1 -9858.624,E2 -9858.624} C_VEL
LIN {X 0,Y 425.321,Z 250.509,A -85,B 0,C 180,E1 -9861.103,E2 -9861.103} C_VEL
LIN {X 0,Y 425.298,Z 250.511,A -85,B 0,C 180,E1 -9864.663,E2 -9864.663} C_VEL
LIN {X 0,Y 425.263,Z 250.514,A -85,B 0,C 180,E1 -9868.072,E2 -9868.072} C_VEL
LIN {X 0,Y 425.334,Z 250.504,A -85,B 0,C 180,E1 -9871.367,E2 -9871.367} C_VEL
LIN {X 0,Y 425.291,Z 250.511,A -85,B 0,C 180,E1 -9874.553,E2 -9874.553} C_VEL
LIN {X 0,Y 425.283,Z 250.511,A -85,B 0,C 180,E1 -9877.66,E2 -9877.66} C_VEL
LIN {X 0,Y 425.357,Z 250.503,A -85,B 0,C 180,E1 -9880.703,E2 -9880.703} C_VEL
LIN {X 0,Y 425.382,Z 250.499,A -85,B 0,C 180,E1 -9883.687,E2 -9883.687} C_VEL
LIN {X 0,Y 425.406,Z 250.496,A -85,B 0,C 180,E1 -9887.597,E2 -9887.597} C_VEL
LIN {X 0,Y 425.436,Z 250.494,A -85,B 0,C 180,E1 -9891.449,E2 -9891.449} C_VEL
LIN {X 0,Y 425.547,Z 250.48,A -85,B 0,C 180,E1 -9894.312,E2 -9894.312} C_VEL
LIN {X 0,Y 425.568,Z 250.476,A -85,B 0,C 180,E1 -9898.106,E2 -9898.106} C_VEL
LIN {X 0,Y 425.695,Z 250.461,A -85,B 0,C 180,E1 -9899.999,E2 -9899.999} C_VEL
LIN {X 0,Y 425.55,Z 250.481,A -85,B 0,C 180,E1 -9902.839,E2 -9902.839} C_VEL
LIN {X 0,Y 425.522,Z 250.483,A -85,B 0,C 180,E1 -9906.644,E2 -9906.644} C_VEL
LIN {X 0,Y 425.425,Z 250.496,A -85,B 0,C 180,E1 -9908.549,E2 -9908.549} C_VEL
LIN {X 0,Y 425.415,Z 250.977,A -85,B 0,C 180,E1 -9909.508,E2 -9909.508} C_VEL
LIN {X 0,Y 425.442,Z 254.395,A -85,B 0,C 180,E1 -9912.4,E2 -9912.4} C_VEL
LIN {X 0,Y 425.205,Z 258.015,A -85,B 0,C 180,E1 -9915.333,E2 -9915.333} C_VEL
LIN {X 0,Y 425.002,Z 261.853,A -85,B 0,C 180,E1 -9918.311,E2 -9918.311} C_VEL
LIN {X 0,Y 424.789,Z 265.856,A -85,B 0,C 180,E1 -9921.344,E2 -9921.344} C_VEL
LIN {X 0,Y 424.676,Z 270.059,A -85,B 0,C 180,E1 -9924.47,E2 -9924.47} C_VEL
LIN {X 0,Y 424.477,Z 274.419,A -85,B 0,C 180,E1 -9927.618,E2 -9927.618} C_VEL
LIN {X 0,Y 424.449,Z 276.299,A -85,B 0,C 180,E1 -9928.966,E2 -9928.966} C_VEL
LIN {X 0,Y 428.019,Z 291.664,A -85,B 0,C 180,E1 -9929.679,E2 -9929.679} C_VEL
LIN {X 0,Y 429.138,Z 299.339,A -85,B 0,C 180,E1 -9930.101,E2 -9930.101} C_VEL
LIN {X 0,Y 428.466,Z 312.379,A -85,B 0,C 180,E1 -9930.892,E2 -9930.892} C_VEL
LIN {X 0,Y 427.835,Z 322.822,A -85,B 0,C 180,E1 -9931.711,E2 -9931.711} C_VEL
LIN {X 0,Y 427.169,Z 333.329,A -85,B 0,C 180,E1 -9932.742,E2 -9932.742} C_VEL
LIN {X 0,Y 426.419,Z 343.177,A -85,B 0,C 180,E1 -9933.937,E2 -9933.937} C_VEL
LIN {X 0,Y 425.756,Z 352.213,A -85,B 0,C 180,E1 -9935.291,E2 -9935.291} C_VEL
LIN {X 0,Y 425.207,Z 359.965,A -85,B 0,C 180,E1 -9936.741,E2 -9936.741} C_VEL
LIN {X 0,Y 424.742,Z 366.682,A -85,B 0,C 180,E1 -9938.329,E2 -9938.329} C_VEL
LIN {X 0,Y 424.479,Z 370.933,A -85,B 0,C 180,E1 -9939.599,E2 -9939.599} C_VEL
LIN {X 0,Y 424.267,Z 374.396,A -85,B 0,C 180,E1 -9940.904,E2 -9940.904} C_VEL
LIN {X 0,Y 424.15,Z 376.238,A -85,B 0,C 180,E1 -9941.788,E2 -9941.788} C_VEL
LIN {X 0,Y 424.069,Z 378.401,A -85,B 0,C 180,E1 -9943.182,E2 -9943.182} C_VEL
LIN {X 0,Y 423.992,Z 379.672,A -85,B 0,C 180,E1 -9944.542,E2 -9944.542} C_VEL
LIN {X 0,Y 423.961,Z 380.105,A -85,B 0,C 180,E1 -9945.876,E2 -9945.876} C_VEL
LIN {X 0,Y 423.92,Z 379.758,A -85,B 0,C 180,E1 -9947.179,E2 -9947.179} C_VEL
LIN {X 0,Y 424.036,Z 378.684,A -85,B 0,C 180,E1 -9948.475,E2 -9948.475} C_VEL
LIN {X 0,Y 424.085,Z 376.925,A -85,B 0,C 180,E1 -9949.737,E2 -9949.737} C_VEL
LIN {X 0,Y 424.236,Z 374.076,A -85,B 0,C 180,E1 -9951.131,E2 -9951.131} C_VEL
LIN {X 0,Y 424.492,Z 369.945,A -85,B 0,C 180,E1 -9952.624,E2 -9952.624} C_VEL
LIN {X 0,Y 424.794,Z 364.369,A -85,B 0,C 180,E1 -9954.16,E2 -9954.16} C_VEL
LIN {X 0,Y 425.209,Z 357.071,A -85,B 0,C 180,E1 -9955.73,E2 -9955.73} C_VEL
LIN {X 0,Y 425.844,Z 348.522,A -85,B 0,C 180,E1 -9957.192,E2 -9957.192} C_VEL
LIN {X 0,Y 426.379,Z 339.981,A -85,B 0,C 180,E1 -9958.372,E2 -9958.372} C_VEL
LIN {X 0,Y 427.048,Z 329.02,A -85,B 0,C 180,E1 -9959.599,E2 -9959.599} C_VEL
LIN {X 0,Y 427.703,Z 318.303,A -85,B 0,C 180,E1 -9960.559,E2 -9960.559} C_VEL
LIN {X 0,Y 428.266,Z 306.62,A -85,B 0,C 180,E1 -9961.382,E2 -9961.382} C_VEL
LIN {X 0,Y 428.763,Z 297.565,A -85,B 0,C 180,E1 -9961.885,E2 -9961.885} C_VEL
LIN {X 0,Y 426.23,Z 284.379,A -85,B 0,C 180,E1 -9962.541,E2 -9962.541} C_VEL
LIN {X 0,Y 424.341,Z 275.676,A -85,B 0,C 180,E1 -9962.886,E2 -9962.886} C_VEL
LIN {X 0,Y 424.431,Z 271.753,A -85,B 0,C 180,E1 -9965.602,E2 -9965.602} C_VEL
LIN {X 0,Y 424.608,Z 267.414,A -85,B 0,C 180,E1 -9968.646,E2 -9968.646} C_VEL
LIN {X 0,Y 424.717,Z 263.167,A -85,B 0,C 180,E1 -9971.676,E2 -9971.676} C_VEL
LIN {X 0,Y 424.871,Z 259.073,A -85,B 0,C 180,E1 -9974.653,E2 -9974.653} C_VEL
LIN {X 0,Y 425.108,Z 255.112,A -85,B 0,C 180,E1 -9977.59,E2 -9977.59} C_VEL
LIN {X 0,Y 425.183,Z 251.301,A -85,B 0,C 180,E1 -9980.486,E2 -9980.486} C_VEL
LIN {X 0,Y 425.262,Z 250.512,A -85,B 0,C 180,E1 -9981.447,E2 -9981.447} C_VEL
LIN {X 0,Y 425.521,Z 250.48,A -85,B 0,C 180,E1 -9984.139,E2 -9984.139} C_VEL
LIN {X 0,Y 424.915,Z 250.559,A -85,B 0,C 180,E1 -9984.928,E2 -9984.928} C_VEL
LIN {X 0,Y 422.105,Z 250.911,A -85,B 0,C 180,E1 -9986.21,E2 -9986.21} C_VEL
LIN {X 0,Y 419.678,Z 251.21,A -85,B 0,C 180,E1 -9987.245,E2 -9987.245} C_VEL
LIN {X 0,Y 418.613,Z 251.341,A -85,B 0,C 180,E1 -9988.045,E2 -9988.045} C_VEL
LIN {X 0,Y 418.515,Z 251.352,A -85,B 0,C 180,E1 -9988.317,E2 -9988.317} C_VEL
LIN {X 0,Y 418.663,Z 251.335,A -85,B 0,C 180,E1 -9990,E2 -9990} C_VEL
LIN {X 0,Y 418.501,Z 251.357,A -85,B 0,C 180,E1 -9992.888,E2 -9992.888} C_VEL
LIN {X 0,Y 418.483,Z 251.358,A -85,B 0,C 180,E1 -9996.751,E2 -9996.751} C_VEL
LIN {X 0,Y 418.35,Z 251.374,A -85,B 0,C 180,E1 -9999.671,E2 -9999.671} C_VEL
LIN {X 0,Y 418.344,Z 251.373,A -85,B 0,C 180,E1 -10003.006,E2 -10003.006} C_VEL
LIN {X 0,Y 418.309,Z 251.378,A -85,B 0,C 180,E1 -10006.739,E2 -10006.739} C_VEL
LIN {X 0,Y 418.292,Z 251.382,A -85,B 0,C 180,E1 -10009.803,E2 -10009.803} C_VEL
LIN {X 0,Y 418.233,Z 251.387,A -85,B 0,C 180,E1 -10012.736,E2 -10012.736} C_VEL
LIN {X 0,Y 418.26,Z 251.388,A -85,B 0,C 180,E1 -10015.904,E2 -10015.904} C_VEL
LIN {X 0,Y 418.264,Z 251.384,A -85,B 0,C 180,E1 -10019.162,E2 -10019.162} C_VEL
LIN {X 0,Y 418.249,Z 251.385,A -85,B 0,C 180,E1 -10022.845,E2 -10022.845} C_VEL
LIN {X 0,Y 418.238,Z 251.388,A -85,B 0,C 180,E1 -10026.239,E2 -10026.239} C_VEL
LIN {X 0,Y 418.255,Z 251.387,A -85,B 0,C 180,E1 -10029.681,E2 -10029.681} C_VEL
LIN {X 0,Y 418.274,Z 251.382,A -85,B 0,C 180,E1 -10032.33,E2 -10032.33} C_VEL
LIN {X 0,Y 418.264,Z 251.386,A -85,B 0,C 180,E1 -10035.115,E2 -10035.115} C_VEL
LIN {X 0,Y 418.282,Z 251.382,A -85,B 0,C 180,E1 -10037.774,E2 -10037.774} C_VEL
LIN {X 0,Y 418.256,Z 251.386,A -85,B 0,C 180,E1 -10041.56,E2 -10041.56} C_VEL
LIN {X 0,Y 418.249,Z 251.388,A -85,B 0,C 180,E1 -10045.16,E2 -10045.16} C_VEL
LIN {X 0,Y 418.236,Z 251.389,A -85,B 0,C 180,E1 -10047.473,E2 -10047.473} C_VEL
LIN {X 0,Y 418.267,Z 251.387,A -85,B 0,C 180,E1 -10050.894,E2 -10050.894} C_VEL
LIN {X 0,Y 418.262,Z 251.383,A -85,B 0,C 180,E1 -10054.097,E2 -10054.097} C_VEL
LIN {X 0,Y 418.229,Z 251.389,A -85,B 0,C 180,E1 -10057.265,E2 -10057.265} C_VEL
LIN {X 0,Y 418.274,Z 251.384,A -85,B 0,C 180,E1 -10060.365,E2 -10060.365} C_VEL
LIN {X 0,Y 418.309,Z 251.378,A -85,B 0,C 180,E1 -10063.406,E2 -10063.406} C_VEL
LIN {X 0,Y 418.338,Z 251.376,A -85,B 0,C 180,E1 -10067,E2 -10067} C_VEL
LIN {X 0,Y 418.335,Z 251.378,A -85,B 0,C 180,E1 -10070.33,E2 -10070.33} C_VEL
LIN {X 0,Y 418.485,Z 251.356,A -85,B 0,C 180,E1 -10073.25,E2 -10073.25} C_VEL
LIN {X 0,Y 418.333,Z 251.374,A -85,B 0,C 180,E1 -10075.183,E2 -10075.183} C_VEL
LIN {X 0,Y 418.538,Z 251.352,A -85,B 0,C 180,E1 -10078.077,E2 -10078.077} C_VEL
LIN {X 0,Y 418.666,Z 251.337,A -85,B 0,C 180,E1 -10080.001,E2 -10080.001} C_VEL
LIN {X 0,Y 418.505,Z 251.354,A -85,B 0,C 180,E1 -10082.889,E2 -10082.889} C_VEL
LIN {X 0,Y 418.488,Z 251.356,A -85,B 0,C 180,E1 -10086.752,E2 -10086.752} C_VEL
LIN {X 0,Y 418.354,Z 251.375,A -85,B 0,C 180,E1 -10089.672,E2 -10089.672} C_VEL
LIN {X 0,Y 418.351,Z 251.373,A -85,B 0,C 180,E1 -10093.007,E2 -10093.007} C_VEL
LIN {X 0,Y 418.309,Z 251.378,A -85,B 0,C 180,E1 -10096.737,E2 -10096.737} C_VEL
LIN {X 0,Y 418.267,Z 251.387,A -85,B 0,C 180,E1 -10099.791,E2 -10099.791} C_VEL
LIN {X 0,Y 418.235,Z 251.387,A -85,B 0,C 180,E1 -10102.737,E2 -10102.737} C_VEL
LIN {X 0,Y 418.268,Z 251.386,A -85,B 0,C 180,E1 -10105.905,E2 -10105.905} C_VEL
LIN {X 0,Y 418.263,Z 251.386,A -85,B 0,C 180,E1 -10109.163,E2 -10109.163} C_VEL
LIN {X 0,Y 418.256,Z 251.385,A -85,B 0,C 180,E1 -10112.845,E2 -10112.845} C_VEL
LIN {X 0,Y 418.245,Z 251.385,A -85,B 0,C 180,E1 -10116.239,E2 -10116.239} C_VEL
LIN {X 0,Y 418.252,Z 251.387,A -85,B 0,C 180,E1 -10119.683,E2 -10119.683} C_VEL
LIN {X 0,Y 418.229,Z 251.387,A -85,B 0,C 180,E1 -10122.322,E2 -10122.322} C_VEL
LIN {X 0,Y 418.236,Z 251.391,A -85,B 0,C 180,E1 -10125.11,E2 -10125.11} C_VEL
LIN {X 0,Y 418.241,Z 251.389,A -85,B 0,C 180,E1 -10127.768,E2 -10127.768} C_VEL
LIN {X 0,Y 418.318,Z 251.592,A -85,B 0,C 180,E1 -10129.698,E2 -10129.698} C_VEL
LIN {X 0,Y 419.216,Z 257.074,A -85,B 0,C 180,E1 -10132.878,E2 -10132.878} C_VEL
LIN {X 0,Y 419.381,Z 261.315,A -85,B 0,C 180,E1 -10135.201,E2 -10135.201} C_VEL
LIN {X 0,Y 419.019,Z 266.886,A -85,B 0,C 180,E1 -10138.108,E2 -10138.108} C_VEL
LIN {X 0,Y 418.532,Z 273.414,A -85,B 0,C 180,E1 -10141.408,E2 -10141.408} C_VEL
LIN {X 0,Y 418.205,Z 279.951,A -85,B 0,C 180,E1 -10144.626,E2 -10144.626} C_VEL
LIN {X 0,Y 417.849,Z 287.583,A -85,B 0,C 180,E1 -10148.283,E2 -10148.283} C_VEL
LIN {X 0,Y 417.534,Z 295.202,A -85,B 0,C 180,E1 -10151.857,E2 -10151.857} C_VEL
LIN {X 0,Y 417.501,Z 297.36,A -85,B 0,C 180,E1 -10152.858,E2 -10152.858} C_VEL
LIN {X 0,Y 419.901,Z 311.451,A -85,B 0,C 180,E1 -10153.4,E2 -10153.4} C_VEL
LIN {X 0,Y 421.432,Z 323.904,A -85,B 0,C 180,E1 -10154.051,E2 -10154.051} C_VEL
LIN {X 0,Y 420.914,Z 335.207,A -85,B 0,C 180,E1 -10154.753,E2 -10154.753} C_VEL
LIN {X 0,Y 420.22,Z 346.036,A -85,B 0,C 180,E1 -10155.605,E2 -10155.605} C_VEL
LIN {X 0,Y 419.486,Z 356.896,A -85,B 0,C 180,E1 -10156.682,E2 -10156.682} C_VEL
LIN {X 0,Y 418.874,Z 366.736,A -85,B 0,C 180,E1 -10157.894,E2 -10157.894} C_VEL
LIN {X 0,Y 418.239,Z 374.806,A -85,B 0,C 180,E1 -10159.103,E2 -10159.103} C_VEL
LIN {X 0,Y 417.768,Z 382.734,A -85,B 0,C 180,E1 -10160.56,E2 -10160.56} C_VEL
LIN {X 0,Y 417.469,Z 388.102,A -85,B 0,C 180,E1 -10161.773,E2 -10161.773} C_VEL
LIN {X 0,Y 417.236,Z 393.349,A -85,B 0,C 180,E1 -10163.229,E2 -10163.229} C_VEL
LIN {X 0,Y 417.123,Z 397.415,A -85,B 0,C 180,E1 -10164.683,E2 -10164.683} C_VEL
LIN {X 0,Y 417.015,Z 400.415,A -85,B 0,C 180,E1 -10166.135,E2 -10166.135} C_VEL
LIN {X 0,Y 417.03,Z 401.873,A -85,B 0,C 180,E1 -10167.102,E2 -10167.102} C_VEL
LIN {X 0,Y 417.058,Z 402.897,A -85,B 0,C 180,E1 -10168.069,E2 -10168.069} C_VEL
LIN {X 0,Y 417.005,Z 403.765,A -85,B 0,C 180,E1 -10170,E2 -10170} C_VEL
LIN {X 0,Y 417.012,Z 403.581,A -85,B 0,C 180,E1 -10170.966,E2 -10170.966} C_VEL
LIN {X 0,Y 417.057,Z 402.981,A -85,B 0,C 180,E1 -10171.931,E2 -10171.931} C_VEL
LIN {X 0,Y 417.029,Z 401.987,A -85,B 0,C 180,E1 -10172.898,E2 -10172.898} C_VEL
LIN {X 0,Y 417.015,Z 400.594,A -85,B 0,C 180,E1 -10173.865,E2 -10173.865} C_VEL
LIN {X 0,Y 417.123,Z 397.659,A -85,B 0,C 180,E1 -10175.317,E2 -10175.317} C_VEL
LIN {X 0,Y 417.236,Z 393.683,A -85,B 0,C 180,E1 -10176.771,E2 -10176.771} C_VEL
LIN {X 0,Y 417.527,Z 387.584,A -85,B 0,C 180,E1 -10178.469,E2 -10178.469} C_VEL
LIN {X 0,Y 417.947,Z 380.918,A -85,B 0,C 180,E1 -10179.925,E2 -10179.925} C_VEL
LIN {X 0,Y 418.513,Z 372.66,A -85,B 0,C 180,E1 -10181.38,E2 -10181.38} C_VEL
LIN {X 0,Y 419.239,Z 364.236,A -85,B 0,C 180,E1 -10182.587,E2 -10182.587} C_VEL
LIN {X 0,Y 419.823,Z 354.54,A -85,B 0,C 180,E1 -10183.731,E2 -10183.731} C_VEL
LIN {X 0,Y 420.591,Z 343.674,A -85,B 0,C 180,E1 -10184.763,E2 -10184.763} C_VEL
LIN {X 0,Y 421.386,Z 332.594,A -85,B 0,C 180,E1 -10185.601,E2 -10185.601} C_VEL
LIN {X 0,Y 421.714,Z 323.708,A -85,B 0,C 180,E1 -10186.147,E2 -10186.147} C_VEL
LIN {X 0,Y 420.083,Z 310.631,A -85,B 0,C 180,E1 -10186.851,E2 -10186.851} C_VEL
LIN {X 0,Y 417.64,Z 298.029,A -85,B 0,C 180,E1 -10187.375,E2 -10187.375} C_VEL
LIN {X 0,Y 417.455,Z 296.641,A -85,B 0,C 180,E1 -10187.453,E2 -10187.453} C_VEL
LIN {X 0,Y 417.731,Z 289.744,A -85,B 0,C 180,E1 -10190.689,E2 -10190.689} C_VEL
LIN {X 0,Y 417.976,Z 284.363,A -85,B 0,C 180,E1 -10193.274,E2 -10193.274} C_VEL
LIN {X 0,Y 418.326,Z 277.957,A -85,B 0,C 180,E1 -10196.436,E2 -10196.436} C_VEL
LIN {X 0,Y 418.803,Z 270.571,A -85,B 0,C 180,E1 -10200.227,E2 -10200.227} C_VEL
LIN {X 0,Y 419.213,Z 265.393,A -85,B 0,C 180,E1 -10203.044,E2 -10203.044} C_VEL
LIN {X 0,Y 419.501,Z 262.217,A -85,B 0,C 180,E1 -10204.823,E2 -10204.823} C_VEL
LIN {X 0,Y 419.322,Z 258.366,A -85,B 0,C 180,E1 -10207.111,E2 -10207.111} C_VEL
LIN {X 0,Y 418.791,Z 254.447,A -85,B 0,C 180,E1 -10209.62,E2 -10209.62} C_VEL
LIN {X 0,Y 418.286,Z 251.384,A -85,B 0,C 180,E1 -10211.741,E2 -10211.741} C_VEL
LIN {X 0,Y 418.237,Z 251.389,A -85,B 0,C 180,E1 -10215.108,E2 -10215.108} C_VEL
LIN {X 0,Y 418.255,Z 251.388,A -85,B 0,C 180,E1 -10217.768,E2 -10217.768} C_VEL
LIN {X 0,Y 418.266,Z 251.389,A -85,B 0,C 180,E1 -10220.616,E2 -10220.616} C_VEL
LIN {X 0,Y 418.244,Z 251.389,A -85,B 0,C 180,E1 -10223.975,E2 -10223.975} C_VEL
LIN {X 0,Y 418.255,Z 251.387,A -85,B 0,C 180,E1 -10227.155,E2 -10227.155} C_VEL
LIN {X 0,Y 418.271,Z 251.385,A -85,B 0,C 180,E1 -10230.838,E2 -10230.838} C_VEL
LIN {X 0,Y 418.267,Z 251.386,A -85,B 0,C 180,E1 -10234.095,E2 -10234.095} C_VEL
LIN {X 0,Y 418.233,Z 251.39,A -85,B 0,C 180,E1 -10237.263,E2 -10237.263} C_VEL
LIN {X 0,Y 418.278,Z 251.385,A -85,B 0,C 180,E1 -10240.363,E2 -10240.363} C_VEL
LIN {X 0,Y 418.311,Z 251.38,A -85,B 0,C 180,E1 -10243.403,E2 -10243.403} C_VEL
LIN {X 0,Y 418.34,Z 251.377,A -85,B 0,C 180,E1 -10246.998,E2 -10246.998} C_VEL
LIN {X 0,Y 418.336,Z 251.378,A -85,B 0,C 180,E1 -10250.327,E2 -10250.327} C_VEL
LIN {X 0,Y 418.487,Z 251.359,A -85,B 0,C 180,E1 -10253.248,E2 -10253.248} C_VEL
LIN {X 0,Y 418.334,Z 251.376,A -85,B 0,C 180,E1 -10255.18,E2 -10255.18} C_VEL
LIN {X 0,Y 418.537,Z 251.352,A -85,B 0,C 180,E1 -10258.074,E2 -10258.074} C_VEL
LIN {X 0,Y 418.664,Z 251.336,A -85,B 0,C 180,E1 -10259.999,E2 -10259.999} C_VEL
LIN {X 0,Y 418.504,Z 251.359,A -85,B 0,C 180,E1 -10262.887,E2 -10262.887} C_VEL
LIN {X 0,Y 418.485,Z 251.36,A -85,B 0,C 180,E1 -10266.75,E2 -10266.75} C_VEL
LIN {X 0,Y 418.389,Z 251.372,A -85,B 0,C 180,E1 -10268.694,E2 -10268.694} C_VEL
LIN {X 0,Y 418.42,Z 253.375,A -85,B 0,C 180,E1 -10270.646,E2 -10270.646} C_VEL
LIN {X 0,Y 418.374,Z 256.162,A -85,B 0,C 180,E1 -10273.022,E2 -10273.022} C_VEL
LIN {X 0,Y 418.1,Z 260.62,A -85,B 0,C 180,E1 -10276.642,E2 -10276.642} C_VEL
LIN {X 0,Y 417.859,Z 264.487,A -85,B 0,C 180,E1 -10279.655,E2 -10279.655} C_VEL
LIN {X 0,Y 417.674,Z 268.562,A -85,B 0,C 180,E1 -10282.767,E2 -10282.767} C_VEL
LIN {X 0,Y 417.571,Z 271.391,A -85,B 0,C 180,E1 -10284.881,E2 -10284.881} C_VEL
LIN {X 0,Y 417.383,Z 276.549,A -85,B 0,C 180,E1 -10288.652,E2 -10288.652} C_VEL
LIN {X 0,Y 420.874,Z 291.165,A -85,B 0,C 180,E1 -10289.339,E2 -10289.339} C_VEL
LIN {X 0,Y 422.349,Z 299.42,A -85,B 0,C 180,E1 -10289.809,E2 -10289.809} C_VEL
LIN {X 0,Y 421.682,Z 312.569,A -85,B 0,C 180,E1 -10290.62,E2 -10290.62} C_VEL
LIN {X 0,Y 420.946,Z 323.805,A -85,B 0,C 180,E1 -10291.521,E2 -10291.521} C_VEL
LIN {X 0,Y 420.184,Z 334.705,A -85,B 0,C 180,E1 -10292.632,E2 -10292.632} C_VEL
LIN {X 0,Y 419.418,Z 344.435,A -85,B 0,C 180,E1 -10293.858,E2 -10293.858} C_VEL
LIN {X 0,Y 418.806,Z 352.363,A -85,B 0,C 180,E1 -10295.08,E2 -10295.08} C_VEL
LIN {X 0,Y 418.23,Z 359.597,A -85,B 0,C 180,E1 -10296.44,E2 -10296.44} C_VEL
LIN {X 0,Y 417.739,Z 366.57,A -85,B 0,C 180,E1 -10298.097,E2 -10298.097} C_VEL
LIN {X 0,Y 417.386,Z 372.024,A -85,B 0,C 180,E1 -10299.779,E2 -10299.779} C_VEL
LIN {X 0,Y 417.169,Z 375.188,A -85,B 0,C 180,E1 -10301.072,E2 -10301.072} C_VEL
LIN {X 0,Y 417.019,Z 377.597,A -85,B 0,C 180,E1 -10302.384,E2 -10302.384} C_VEL
LIN {X 0,Y 416.955,Z 379.263,A -85,B 0,C 180,E1 -10303.713,E2 -10303.713} C_VEL
LIN {X 0,Y 416.883,Z 380.15,A -85,B 0,C 180,E1 -10305.075,E2 -10305.075} C_VEL
LIN {X 0,Y 416.83,Z 380.232,A -85,B 0,C 180,E1 -10306.467,E2 -10306.467} C_VEL
LIN {X 0,Y 416.874,Z 379.477,A -85,B 0,C 180,E1 -10307.882,E2 -10307.882} C_VEL
LIN {X 0,Y 416.964,Z 377.814,A -85,B 0,C 180,E1 -10309.328,E2 -10309.328} C_VEL
LIN {X 0,Y 417.108,Z 375.139,A -85,B 0,C 180,E1 -10310.809,E2 -10310.809} C_VEL
LIN {X 0,Y 417.348,Z 371.318,A -85,B 0,C 180,E1 -10312.32,E2 -10312.32} C_VEL
LIN {X 0,Y 417.695,Z 365.943,A -85,B 0,C 180,E1 -10313.922,E2 -10313.922} C_VEL
LIN {X 0,Y 418.08,Z 359.378,A -85,B 0,C 180,E1 -10315.454,E2 -10315.454} C_VEL
LIN {X 0,Y 418.547,Z 352.566,A -85,B 0,C 180,E1 -10316.734,E2 -10316.734} C_VEL
LIN {X 0,Y 419.23,Z 343.423,A -85,B 0,C 180,E1 -10318.126,E2 -10318.126} C_VEL
LIN {X 0,Y 419.886,Z 332.708,A -85,B 0,C 180,E1 -10319.443,E2 -10319.443} C_VEL
LIN {X 0,Y 420.55,Z 322.62,A -85,B 0,C 180,E1 -10320.432,E2 -10320.432} C_VEL
LIN {X 0,Y 421.211,Z 310.694,A -85,B 0,C 180,E1 -10321.362,E2 -10321.362} C_VEL
LIN {X 0,Y 421.877,Z 298.999,A -85,B 0,C 180,E1 -10322.063,E2 -10322.063} C_VEL
LIN {X 0,Y 419.521,Z 286.138,A -85,B 0,C 180,E1 -10322.738,E2 -10322.738} C_VEL
LIN {X 0,Y 417.274,Z 275.872,A -85,B 0,C 180,E1 -10323.153,E2 -10323.153} C_VEL
LIN {X 0,Y 417.371,Z 271.578,A -85,B 0,C 180,E1 -10326.164,E2 -10326.164} C_VEL
LIN {X 0,Y 417.568,Z 267.169,A -85,B 0,C 180,E1 -10329.302,E2 -10329.302} C_VEL
LIN {X 0,Y 417.714,Z 262.95,A -85,B 0,C 180,E1 -10332.372,E2 -10332.372} C_VEL
LIN {X 0,Y 417.839,Z 258.872,A -85,B 0,C 180,E1 -10335.387,E2 -10335.387} C_VEL
LIN {X 0,Y 418.088,Z 254.928,A -85,B 0,C 180,E1 -10338.363,E2 -10338.363} C_VEL
LIN {X 0,Y 418.14,Z 252.39,A -85,B 0,C 180,E1 -10340.324,E2 -10340.324} C_VEL
LIN {X 0,Y 418.19,Z 251.394,A -85,B 0,C 180,E1 -10341.301,E2 -10341.301} C_VEL
LIN {X 0,Y 418.488,Z 251.357,A -85,B 0,C 180,E1 -10344.152,E2 -10344.152} C_VEL
LIN {X 0,Y 418.535,Z 251.351,A -85,B 0,C 180,E1 -10348.076,E2 -10348.076} C_VEL
LIN {X 0,Y 418.515,Z 251.352,A -85,B 0,C 180,E1 -10348.317,E2 -10348.317} C_VEL
LIN {X 0,Y 417.824,Z 251.44,A -85,B 0,C 180,E1 -10349.12,E2 -10349.12} C_VEL
LIN {X 0,Y 414.979,Z 251.795,A -85,B 0,C 180,E1 -10350.426,E2 -10350.426} C_VEL
LIN {X 0,Y 412.582,Z 252.091,A -85,B 0,C 180,E1 -10351.48,E2 -10351.48} C_VEL
LIN {X 0,Y 411.548,Z 252.224,A -85,B 0,C 180,E1 -10352.295,E2 -10352.295} C_VEL
LIN {X 0,Y 411.46,Z 252.231,A -85,B 0,C 180,E1 -10352.571,E2 -10352.571} C_VEL
LIN {X 0,Y 411.465,Z 252.232,A -85,B 0,C 180,E1 -10355.882,E2 -10355.882} C_VEL
LIN {X 0,Y 411.471,Z 252.23,A -85,B 0,C 180,E1 -10357.854,E2 -10357.854} C_VEL
LIN {X 0,Y 411.289,Z 252.254,A -85,B 0,C 180,E1 -10361.833,E2 -10361.833} C_VEL
LIN {X 0,Y 411.256,Z 252.257,A -85,B 0,C 180,E1 -10364.853,E2 -10364.853} C_VEL
LIN {X 0,Y 411.243,Z 252.262,A -85,B 0,C 180,E1 -10367.915,E2 -10367.915} C_VEL
LIN {X 0,Y 411.205,Z 252.263,A -85,B 0,C 180,E1 -10371.033,E2 -10371.033} C_VEL
LIN {X 0,Y 411.218,Z 252.264,A -85,B 0,C 180,E1 -10374.216,E2 -10374.216} C_VEL
LIN {X 0,Y 411.249,Z 252.26,A -85,B 0,C 180,E1 -10377.478,E2 -10377.478} C_VEL
LIN {X 0,Y 411.189,Z 252.265,A -85,B 0,C 180,E1 -10380.847,E2 -10380.847} C_VEL
LIN {X 0,Y 411.195,Z 252.265,A -85,B 0,C 180,E1 -10384.334,E2 -10384.334} C_VEL
LIN {X 0,Y 411.194,Z 252.266,A -85,B 0,C 180,E1 -10387.973,E2 -10387.973} C_VEL
LIN {X 0,Y 411.199,Z 252.266,A -85,B 0,C 180,E1 -10391.236,E2 -10391.236} C_VEL
LIN {X 0,Y 411.226,Z 252.26,A -85,B 0,C 180,E1 -10394.483,E2 -10394.483} C_VEL
LIN {X 0,Y 411.218,Z 252.264,A -85,B 0,C 180,E1 -10397.298,E2 -10397.298} C_VEL
LIN {X 0,Y 411.221,Z 252.262,A -85,B 0,C 180,E1 -10400.778,E2 -10400.778} C_VEL
LIN {X 0,Y 411.19,Z 252.264,A -85,B 0,C 180,E1 -10404.472,E2 -10404.472} C_VEL
LIN {X 0,Y 411.197,Z 252.266,A -85,B 0,C 180,E1 -10406.874,E2 -10406.874} C_VEL
LIN {X 0,Y 411.231,Z 252.261,A -85,B 0,C 180,E1 -10410.643,E2 -10410.643} C_VEL
LIN {X 0,Y 411.229,Z 252.26,A -85,B 0,C 180,E1 -10413.62,E2 -10413.62} C_VEL
LIN {X 0,Y 411.194,Z 252.268,A -85,B 0,C 180,E1 -10416.853,E2 -10416.853} C_VEL
LIN {X 0,Y 411.206,Z 252.262,A -85,B 0,C 180,E1 -10420.051,E2 -10420.051} C_VEL
LIN {X 0,Y 411.255,Z 252.258,A -85,B 0,C 180,E1 -10423.132,E2 -10423.132} C_VEL
LIN {X 0,Y 411.297,Z 252.253,A -85,B 0,C 180,E1 -10426.897,E2 -10426.897} C_VEL
LIN {X 0,Y 411.287,Z 252.255,A -85,B 0,C 180,E1 -10430.162,E2 -10430.162} C_VEL
LIN {X 0,Y 411.449,Z 252.233,A -85,B 0,C 180,E1 -10433.134,E2 -10433.134} C_VEL
LIN {X 0,Y 411.304,Z 252.25,A -85,B 0,C 180,E1 -10435.1,E2 -10435.1} C_VEL
LIN {X 0,Y 411.507,Z 252.227,A -85,B 0,C 180,E1 -10438.044,E2 -10438.044} C_VEL
LIN {X 0,Y 411.635,Z 252.212,A -85,B 0,C 180,E1 -10440.001,E2 -10440.001} C_VEL
LIN {X 0,Y 411.461,Z 252.231,A -85,B 0,C 180,E1 -10442.938,E2 -10442.938} C_VEL
LIN {X 0,Y 411.455,Z 252.232,A -85,B 0,C 180,E1 -10446.868,E2 -10446.868} C_VEL
LIN {X 0,Y 411.303,Z 252.253,A -85,B 0,C 180,E1 -10449.84,E2 -10449.84} C_VEL
LIN {X 0,Y 411.309,Z 252.25,A -85,B 0,C 180,E1 -10453.11,E2 -10453.11} C_VEL
LIN {X 0,Y 411.254,Z 252.256,A -85,B 0,C 180,E1 -10456.89,E2 -10456.89} C_VEL
LIN {X 0,Y 411.228,Z 252.263,A -85,B 0,C 180,E1 -10459.988,E2 -10459.988} C_VEL
LIN {X 0,Y 411.201,Z 252.265,A -85,B 0,C 180,E1 -10463.149,E2 -10463.149} C_VEL
LIN {X 0,Y 411.236,Z 252.258,A -85,B 0,C 180,E1 -10466.382,E2 -10466.382} C_VEL
LIN {X 0,Y 411.199,Z 252.266,A -85,B 0,C 180,E1 -10469.714,E2 -10469.714} C_VEL
LIN {X 0,Y 411.205,Z 252.265,A -85,B 0,C 180,E1 -10473.157,E2 -10473.157} C_VEL
LIN {X 0,Y 411.193,Z 252.264,A -85,B 0,C 180,E1 -10476.554,E2 -10476.554} C_VEL
LIN {X 0,Y 411.215,Z 252.263,A -85,B 0,C 180,E1 -10479.729,E2 -10479.729} C_VEL
LIN {X 0,Y 411.173,Z 252.27,A -85,B 0,C 180,E1 -10483.135,E2 -10483.135} C_VEL
LIN {X 0,Y 411.169,Z 252.268,A -85,B 0,C 180,E1 -10485.882,E2 -10485.882} C_VEL
LIN {X 0,Y 411.224,Z 252.37,A -85,B 0,C 180,E1 -10489.431,E2 -10489.431} C_VEL
LIN {X 0,Y 412.046,Z 256.866,A -85,B 0,C 180,E1 -10492.119,E2 -10492.119} C_VEL
LIN {X 0,Y 412.402,Z 261.79,A -85,B 0,C 180,E1 -10494.886,E2 -10494.886} C_VEL
LIN {X 0,Y 412.07,Z 266.702,A -85,B 0,C 180,E1 -10497.504,E2 -10497.504} C_VEL
LIN {X 0,Y 411.625,Z 272.575,A -85,B 0,C 180,E1 -10500.549,E2 -10500.549} C_VEL
LIN {X 0,Y 411.176,Z 279.756,A -85,B 0,C 180,E1 -10504.161,E2 -10504.161} C_VEL
LIN {X 0,Y 410.799,Z 287.369,A -85,B 0,C 180,E1 -10507.891,E2 -10507.891} C_VEL
LIN {X 0,Y 410.541,Z 293.888,A -85,B 0,C 180,E1 -10511.019,E2 -10511.019} C_VEL
LIN {X 0,Y 410.441,Z 297.333,A -85,B 0,C 180,E1 -10512.592,E2 -10512.592} C_VEL
LIN {X 0,Y 412.739,Z 310.831,A -85,B 0,C 180,E1 -10513.113,E2 -10513.113} C_VEL
LIN {X 0,Y 414.457,Z 324.022,A -85,B 0,C 180,E1 -10513.816,E2 -10513.816} C_VEL
LIN {X 0,Y 414.167,Z 332.949,A -85,B 0,C 180,E1 -10514.373,E2 -10514.373} C_VEL
LIN {X 0,Y 413.411,Z 344.048,A -85,B 0,C 180,E1 -10515.227,E2 -10515.227} C_VEL
LIN {X 0,Y 412.643,Z 355.045,A -85,B 0,C 180,E1 -10516.29,E2 -10516.29} C_VEL
LIN {X 0,Y 412.038,Z 364.602,A -85,B 0,C 180,E1 -10517.439,E2 -10517.439} C_VEL
LIN {X 0,Y 411.34,Z 372.994,A -85,B 0,C 180,E1 -10518.669,E2 -10518.669} C_VEL
LIN {X 0,Y 410.811,Z 381.21,A -85,B 0,C 180,E1 -10520.15,E2 -10520.15} C_VEL
LIN {X 0,Y 410.425,Z 387.824,A -85,B 0,C 180,E1 -10521.631,E2 -10521.631} C_VEL
LIN {X 0,Y 410.169,Z 393.089,A -85,B 0,C 180,E1 -10523.111,E2 -10523.111} C_VEL
LIN {X 0,Y 410.019,Z 397.169,A -85,B 0,C 180,E1 -10524.59,E2 -10524.59} C_VEL
